// TwinCAT 3 PLC project RobustSolutionFramework
// Title: RobustSolution
// Company: BATW
// Author: BATW
// ProjectVersion: 1.0.0.1
// ProgramVersion: 3.1.4026.24
// libraries:
//   Tc2_MC2, * (Beckhoff Automation GmbH)
//   Tc2_Standard, * (Beckhoff Automation GmbH)
//   Tc2_System, * (Beckhoff Automation GmbH)
//   Tc2_Utilities, * (Beckhoff Automation GmbH)
//   Tc3_JsonXml, * (Beckhoff Automation GmbH)
// project tree:
//   Configuration/DUTs/ E_AlarmOperator.TcDUT, E_ConfigDataType.TcDUT (not stored), E_ConfigValueError.TcDUT, E_LinkPhase.TcDUT, E_ModuleType.TcDUT (not stored), T_ModuleTypeName.TcDUT, E_VariableAccess.TcDUT (not stored), ST_ConfigRawValue.TcDUT, ST_ReferenceBindingFileConfig.TcDUT (not stored), ST_ConfigAlarmInfo.TcDUT, ST_ConfigVariableInfo.TcDUT, ST_RuntimeAlarmBinding.TcDUT, ST_RuntimeVariableBinding.TcDUT, ST_LinkVariableNode.TcDUT (not stored), ST_MappingFileConfig.TcDUT (not stored), ST_ModuleFileConfig.TcDUT (not stored), ST_ModuleRuntimeConfig.TcDUT (not stored), ST_SystemFileConfig.TcDUT (not stored), ST_VariableLink.TcDUT
//   Configuration/POUs/ F_AlarmConditionMet.TcPOU (not stored), F_ConfigDataTypeSize.TcPOU (not stored), F_ConfigDataTypeToDescriptor.TcPOU, F_ConfigValueErrorMessage.TcPOU (not stored), FB_ConfigValueSnapshotReader.TcPOU, FB_ModuleTypeRegistry.TcPOU (not stored), FB_ReferenceManager.TcPOU (not stored), FB_ModuleReferenceBindingContext.TcPOU, FB_LinkVariableManager.TcPOU (not stored), FB_ModuleConfigurationManager.TcPOU (not stored), FB_ApplicationConfigRoot.TcPOU (not stored)
//   Configuration/Interfaces/ I_AdsSymbolProvider.TcIO (not stored), I_ModuleReferenceBindings.TcIO (not stored), I_ModuleConfigurationAdapter.TcIO (not stored), I_VariableNodeReader.TcIO (not stored)
//   DUTs/Contracts/Alarm/ E_Severity.TcDUT, ST_ExtAlarm.TcDUT
//   DUTs/Contracts/Descriptor/ E_DescriptorType.TcDUT, ST_ExtDescriptor.TcDUT (not stored)
//   DUTs/Contracts/System/ ST_SystemContext.TcDUT (not stored)
//   DUTs/Infrastructure/EL Modules/ ST_EL1889Ex.TcDUT (not stored), ST_EL2809Ex.TcDUT (not stored), ST_EL3602Ex.TcDUT (not stored)
//   DUTs/Infrastructure/ ST_ReserveForGetSymbolNameByAddrress.TcDUT
//   DUTs/Module/Alarm/ E_AlarmAckCommand.TcDUT (not stored), E_AlarmAckError.TcDUT (not stored), ST_AlarmAckRequest.TcDUT (not stored), ST_AlarmLifecycleState.TcDUT, ST_ModuleAlarmStatus.TcDUT (not stored)
//   DUTs/Module/Contract/ ST_ModuleCtrl.TcDUT, ST_ModuleDataStatus.TcDUT, ST_ModuleStatus.TcDUT, ST_ModuleVariableStatus.TcDUT (not stored), ST_Module_CtrlStatus_Base.TcDUT (not stored)
//   DUTs/Module/ServiceCoordination/ E_CompositeOwnershipState.TcDUT (not stored), E_ServiceCallSubmitResult.TcDUT (not stored), E_ServiceInternalCommandState.TcDUT, E_ServiceRegistrationError.TcDUT (not stored), ST_ServiceExecutionSnapshot.TcDUT (not stored), ST_ServiceRegistrationEntry.TcDUT (not stored)
//   DUTs/Service/Composite/ E_CompositeServiceErrorCode.TcDUT (not stored)
//   DUTs/Service/Contracts/ E_ServiceCompletionBehavior.TcDUT, ST_EmptyServiceParam.TcDUT, ST_ServiceContext.TcDUT, ST_ServiceCtrl.TcDUT (not stored), ST_ServiceDataStatus.TcDUT (not stored), ST_ServiceExecuteSubStateRecord.TcDUT, ST_ServiceExecuteSubStateStatus.TcDUT, ST_ServiceStatus.TcDUT
//   DUTs/Wafer Transfer/ E_MaterialOperateState.TcDUT, ST_MaterialContext.TcDUT, ST_WaferStatus.TcDUT
//   GVLs/ Param_Config.TcGVL
//   POUs/00_BaseUnit/Base/ FB_BaseUnit.TcPOU (not stored), T_ResourceOwnerId.TcDUT (not stored)
//   POUs/00_BaseUnit/ FB_Axis_BaseUnit.TcPOU (not stored)
//   POUs/00_BaseUnit/Interfaces/ I_Axis_BaseUnit.TcIO (not stored), I_BaseUnit.TcIO (not stored), I_ResourceLock.TcIO
//   POUs/10_Module/ FB_ModuleAlarmManager.TcPOU (not stored), FB_ModuleBase.TcPOU (not stored), FB_ServiceCoordinator.TcPOU, FB_ServiceCaller.TcPOU (not stored)
//   POUs/20_Service/ E_FrameworkServiceErrorCode.TcDUT, FB_CompositeServiceBase.TcPOU, FB_ServiceBase.TcPOU
//   POUs/20_Service/Material Service/ E_SetMaterialCmdType.TcDUT, FB_SetMaterialService.TcPOU, ST_MaterialParam.TcDUT
//   POUs/ FB_UtcClock.TcPOU
//   POUs/30_PackML_Base/DUTs/ E_PackMLCommand.TcDUT (not stored), E_PackMLErrorID.TcDUT (not stored), E_PackMLHookResult.TcDUT (not stored), E_PackMLMode.TcDUT (not stored), E_PackMLState.TcDUT, ST_PML_Base_In.TcDUT, ST_PML_Base_Out.TcDUT, T_PackMLMode.TcDUT (not stored)
//   POUs/30_PackML_Base/ FB_PackMLBase.TcPOU (not stored), FB_PackMLModeSet.TcPOU
//   POUs/30_PackML_Base/Utilities/ F_PackMLCommandToString.TcPOU (not stored), F_PackMLErrorIDToString.TcPOU (not stored), F_PackMLModeToString.TcPOU (not stored), F_PackMLStateToString.TcPOU (not stored)
// real-time tasks:
//   TASK UnitTest Task: cycle T#10ms, priority 21, ADS port 351
//   TASK DemoProject Task: cycle T#10ms, priority 22, ADS port 352
// motion (NC):
//   TASK NC-Task 1 SAF: cycle T#2ms, priority 4, ADS port 501
//   TASK NC-Task 1 SVB: cycle T#10ms, priority 8, ADS port 511
//   AXIS Axis 1 (id 1)
//     OtherSettings: AllowMotionCmdToSlave=true
//     encoder EncType=1
//     drive DrvType=5
//       Analog: TorqueSetpointScale=10, ScaleFactorActTorque=0.1
//       TimeComp: TaskDelayCycles=1
//     controller CtrType=1
//       CtrPara: PriorControlFactor=1
//         Observer: BandWidth=20
//   AXIS Axis 2 (id 2)
//     OtherSettings: AllowMotionCmdToSlave=true
//     encoder EncType=1
//     drive DrvType=5
//       Analog: TorqueSetpointScale=10, ScaleFactorActTorque=0.1
//       TimeComp: TaskDelayCycles=1
//     controller CtrType=1
//       CtrPara: PriorControlFactor=1
//         Observer: BandWidth=20
// variable links:
//   RobustSolutionDemoProject/RobustSolutionDemoProject Instance <-> NC-Task 1 SAF/Axes/Axis 1
//     PlcTask Inputs/GVL_IO.NC_Axis1._Axis.NcToPlc <-> Outputs/ToPlc
//     PlcTask Outputs/GVL_IO.NC_Axis1._Axis.PlcToNc <-> Inputs/FromPlc
//   RobustSolutionDemoProject/RobustSolutionDemoProject Instance <-> NC-Task 1 SAF/Axes/Axis 2
//     PlcTask Inputs/GVL_IO.NC_Axis2._Axis.NcToPlc <-> Outputs/ToPlc
//     PlcTask Outputs/GVL_IO.NC_Axis2._Axis.PlcToNc <-> Inputs/FromPlc

// ---- Configuration/DUTs/E_AlarmOperator.TcDUT
{attribute 'qualified_only'}
{attribute 'strict'}
{attribute 'to_string'}
TYPE E_AlarmOperator :
(
	Invalid := 0,
    GreaterThan,
    LessThan,
    Equal,
    GreaterOrEqual,
    LessOrEqual
);
END_TYPE

// ---- Configuration/DUTs/E_ConfigValueError.TcDUT
{attribute 'qualified_only'}
{attribute 'strict'}
{attribute 'to_string'}
TYPE E_ConfigValueError :
(
	None := 0,
	// FB_ConfigValueSnapshotReader cannot access the injected node reader.
	ReaderUnavailable := 16#7100,
	// The configured VariableList and AlarmList exceed the snapshot capacity.
	SourceCapacityExceeded := 16#7101,
	// FB_LinkVariableManager received an unknown or expired opaque handle.
	InvalidNodeHandle := 16#7201,
	// The registered node cannot be used as a configured value source.
	NodeReadNotAllowed := 16#7202,
	// The registered node no longer has a valid data address.
	InvalidNodeAddress := 16#7203,
	// Config metadata and registered node metadata do not describe the same type.
	NodeDataTypeMismatch := 16#7204,
	// The registered size is zero or exceeds ST_ConfigRawValue.Data.
	InvalidNodeSize := 16#7205
)UDINT;
END_TYPE

// ---- Configuration/DUTs/E_LinkPhase.TcDUT
{attribute 'qualified_only'}
{attribute 'strict'}
TYPE E_LinkPhase :
(
	InputToModule := 1,
	ModuleToOutput
);
END_TYPE

// ---- Configuration/DUTs/T_ModuleTypeName.TcDUT
TYPE T_ModuleTypeName : STRING(16);
END_TYPE

// ---- Configuration/DUTs/ST_ConfigRawValue.TcDUT
{attribute 'pack_mode' := '1'}
TYPE ST_ConfigRawValue :
STRUCT
	Data : ARRAY[0..Param_Config.MaxConfigValueSize - 1] OF BYTE;
END_STRUCT
END_TYPE

// ---- Configuration/DUTs/ST_ConfigAlarmInfo.TcDUT
TYPE ST_ConfigAlarmInfo :
STRUCT
	Source : STRING(255);
	DataType : E_ConfigDataType;
	Operator : E_AlarmOperator;
	Threshold : LREAL;
	Tolerance : LREAL;
	MainErrorId : UDINT;
	SourceErrorId : UDINT;
	Message : STRING(80);
	Severity : E_Severity;
END_STRUCT
END_TYPE

// ---- Configuration/DUTs/ST_ConfigVariableInfo.TcDUT
TYPE ST_ConfigVariableInfo :
STRUCT
	Source : STRING(255);
	Id : UDINT;
	Name : STRING(30);
	Unit : STRING(10);
	DataType : E_ConfigDataType;
END_STRUCT
END_TYPE

// ---- Configuration/DUTs/ST_RuntimeAlarmBinding.TcDUT
TYPE ST_RuntimeAlarmBinding :
STRUCT
	Definition : ST_ConfigAlarmInfo;
	NodeHandle : UINT;
END_STRUCT
END_TYPE

// ---- Configuration/DUTs/ST_RuntimeVariableBinding.TcDUT
TYPE ST_RuntimeVariableBinding :
STRUCT
	Definition : ST_ConfigVariableInfo;
	NodeHandle : UINT;
END_STRUCT
END_TYPE

// ---- Configuration/DUTs/ST_VariableLink.TcDUT
TYPE ST_VariableLink :
STRUCT
	SourceAddress : PVOID;
	TargetAddress : PVOID;
	SourceSize : UDINT;
	TargetSize : UDINT;
	SourceDataType : E_ConfigDataType;
	TargetDataType : E_ConfigDataType;
	Phase : E_LinkPhase;
	HasTransform : BOOL;
	Scale : LREAL;
	Offset : LREAL;
END_STRUCT
END_TYPE

// ---- DUTs/Contracts/Alarm/E_Severity.TcDUT
{attribute 'qualified_only'}
{attribute 'strict'}
{attribute 'to_string'}
TYPE E_Severity :
(
	Alarm := 1,
	Warning
);
END_TYPE

// ---- DUTs/Contracts/Alarm/ST_ExtAlarm.TcDUT
TYPE ST_ExtAlarm :
STRUCT
	ModuleId : UDINT;
	ServiceId : UDINT;
	MainErrorId : UDINT;
	SourceErrorId : UDINT;
	Message : STRING;
	Path : STRING(255);
	Severity : E_Severity;
	DateTime : STRING(20);	// First occurrence of the current alarm lifecycle. ex: YYYYMMDDHHMMSSUUU
	Active : BOOL;
	Acknowledged : BOOL;
	OccurrenceCount : UDINT;
END_STRUCT
END_TYPE

// ---- DUTs/Contracts/Descriptor/E_DescriptorType.TcDUT
{attribute 'qualified_only'}
{attribute 'strict'}
{attribute 'to_string'}
TYPE E_DescriptorType :
(
	Integer_32bit := 1,	// TwinCAT DINT, CSharp int
	Float_32bit,		// TwinCAT REAL, CSharp float
	String_80byte,
	DateTime,	// ex: YYYYMMDDHHMMSSUU
	Boolean,
	Unsigned_32bit,
	Float_64bit
);
END_TYPE

// ---- DUTs/Infrastructure/ST_ReserveForGetSymbolNameByAddrress.TcDUT
TYPE ST_ReserveForGetSymbolNameByAddrress :
STRUCT
	//If structures with a single variable are used, the data type cannot be read correctly using this method.
	//The size and address information cannot be used to distinguish between the structure itself and the individual variables.
	//https://infosys.beckhoff.com/content/1033/tcplclib_tc3_jsonxml/4220928907.html?id=4536537886268406375
	_Reserve : BOOL;
END_STRUCT
END_TYPE

// ---- DUTs/Module/Alarm/ST_AlarmLifecycleState.TcDUT
TYPE ST_AlarmLifecycleState :
STRUCT
	Latched : BOOL;
	PreviousActive : BOOL;
	SeenThisCycle : BOOL;
	Alarm : ST_ExtAlarm;
END_STRUCT
END_TYPE

// ---- DUTs/Module/Contract/ST_ModuleCtrl.TcDUT
TYPE ST_ModuleCtrl :
STRUCT
	RequestId : UDINT;
	PackMLIn : ST_PML_Base_In;
	
	AlarmAckRequest : ST_AlarmAckRequest;
END_STRUCT
END_TYPE

// ---- DUTs/Module/Contract/ST_ModuleDataStatus.TcDUT
TYPE ST_ModuleDataStatus :
STRUCT
	PublishedCount : UINT;
	Overflow : BOOL;
	DuplicateId : UDINT;
END_STRUCT
END_TYPE

// ---- DUTs/Module/Contract/ST_ModuleStatus.TcDUT
TYPE ST_ModuleStatus :
STRUCT
	ModuleId : UDINT;
	Enabled : BOOL;
	IsControlSourceAlive : BOOL;
	ModuleType : STRING(16);
	
	ResponseId : UDINT;
	PackMLOut : ST_PML_Base_Out;
	
	Alarm : ST_ModuleAlarmStatus;
	
	Data : ST_ModuleDataStatus;
	Variable : ST_ModuleVariableStatus;
	
	// Array index is storage only; EndpointId is the external identity.
	WaferStatusList : ARRAY [1..Param_Config.MaxTransferEndpoint] OF ST_WaferStatus;
END_STRUCT
END_TYPE

// ---- DUTs/Module/ServiceCoordination/E_ServiceInternalCommandState.TcDUT
{attribute 'qualified_only'}
{attribute 'strict'}
{attribute 'to_string'}
TYPE E_ServiceInternalCommandState :
(
	None := 0,
	Queued := 1,
	RequestHigh := 2,
	Accepted := 3,
	Rejected := 4,
	Cancelled := 5
) UDINT;
END_TYPE

// ---- DUTs/Service/Contracts/E_ServiceCompletionBehavior.TcDUT
{attribute 'qualified_only'}
{attribute 'strict'}
{attribute 'to_string'}
TYPE E_ServiceCompletionBehavior :
(
	Unknown := 0,
	NaturalCompletion := 1,
	ExecuteUntilExternalStop := 2
) UDINT;
END_TYPE

// ---- DUTs/Service/Contracts/ST_EmptyServiceParam.TcDUT
TYPE ST_EmptyServiceParam :
STRUCT
	bDummyValue : BOOL;	// To avoid 0 size check error during Service Coordinator Registration
END_STRUCT
END_TYPE

// ---- DUTs/Service/Contracts/ST_ServiceContext.TcDUT
TYPE ST_ServiceContext :
STRUCT
	ModuleId : UDINT;
	// UTC timestamp formatted as YYYYMMDDHHMMSSUUU.
	UtcDateTime : STRING(20);
END_STRUCT
END_TYPE

// ---- DUTs/Service/Contracts/ST_ServiceExecuteSubStateRecord.TcDUT
TYPE ST_ServiceExecuteSubStateRecord :
STRUCT
	Step : UDINT;
	Name : STRING(80);
	// UTC timestamp formatted as YYYYMMDDHHMMSSUUU.
	StartTimestamp : STRING(20);
	// Empty while this occurrence is still active.
	EndTimestamp : STRING(20);
END_STRUCT
END_TYPE

// ---- DUTs/Service/Contracts/ST_ServiceExecuteSubStateStatus.TcDUT
TYPE ST_ServiceExecuteSubStateStatus :
STRUCT
	// Zero whenever the Service is not executing or exposes no substate.
	CurrentStep : UDINT;
	RecordCount : UINT;
	// The first records are preserved when capacity is exhausted.
	Overflow : BOOL;
	Records : ARRAY[1..Param_Config.MaxExecuteSubStateRecords] OF ST_ServiceExecuteSubStateRecord;
END_STRUCT
END_TYPE

// ---- DUTs/Service/Contracts/ST_ServiceStatus.TcDUT
TYPE ST_ServiceStatus :
STRUCT
	ResponseId : UDINT;
	PackMLOut : ST_PML_Base_Out;
	ExecuteSubState : ST_ServiceExecuteSubStateStatus;
	CompletionBehavior : E_ServiceCompletionBehavior;
	ServiceId : UDINT;
	ErrorList : ARRAY[1..Param_Config.MaxServiceError] OF ST_ExtAlarm;
	Data : ST_ServiceDataStatus;
END_STRUCT
END_TYPE

// ---- DUTs/Wafer Transfer/E_MaterialOperateState.TcDUT
{attribute 'qualified_only'}
{attribute 'strict'}
{attribute 'to_string'}
TYPE E_MaterialOperateState :
(
	NotApplicable := 0,
	Pending,
	Processing,
	Completed,
	Failed
);
END_TYPE

// ---- DUTs/Wafer Transfer/ST_MaterialContext.TcDUT
TYPE ST_MaterialContext :
STRUCT
	Id : STRING(80);
	OperationState : E_MaterialOperateState;
	// Add other information of wafer...
END_STRUCT
END_TYPE

// ---- DUTs/Wafer Transfer/ST_WaferStatus.TcDUT
TYPE ST_WaferStatus :
STRUCT
	// Managed by module
	// Non-zero and unique within one Module; array index is storage only.
	EndpointId : UDINT;
	EndpointName : STRING(80);
	MaterialContext : ST_MaterialContext;
END_STRUCT
END_TYPE

// ---- POUs/20_Service/E_FrameworkServiceErrorCode.TcDUT
{attribute 'qualified_only'}
{attribute 'strict'}
{attribute 'to_string'}
TYPE E_FrameworkServiceErrorCode :
(
	// Set material service
	None := 0,
	SetMaterial_InvalidCmd := 900,
	SetMaterial_TaEpIdRequired := 901,
	SetMaterial_TaEpNotFound := 902,
	SetMaterial_DuplicateTaEpId := 903
) UDINT;
END_TYPE

// ---- POUs/20_Service/Material Service/E_SetMaterialCmdType.TcDUT
{attribute 'qualified_only'}
{attribute 'strict'}
{attribute 'to_string'}
TYPE E_SetMaterialCmdType :
(
	Modify:= 1,
	Clear,
	ClearAll
);
END_TYPE

// ---- POUs/20_Service/Material Service/ST_MaterialParam.TcDUT
TYPE ST_MaterialParam :
STRUCT
	CmdType : E_SetMaterialCmdType;
	TargetEndpointId : UDINT;
	
	// Material context
	MaterialId : STRING(80);
	MaterialOperateState : E_MaterialOperateState;
END_STRUCT
END_TYPE

// ---- POUs/30_PackML_Base/DUTs/E_PackMLState.TcDUT
{attribute 'qualified_only'}
TYPE E_PackMLState :
(
	Undefined		:= 0,
	Clearing		:= 1,
	Stopped			:= 2,
	Starting		:= 3,
	Idle			:= 4,
	Suspended		:= 5,
	Execute			:= 6,
	Stopping		:= 7,
	Aborting		:= 8,
	Aborted			:= 9,
	Holding			:= 10,
	Held			:= 11,
	Unholding		:= 12,
	Suspending		:= 13,
	Unsuspending	:= 14,
	Resetting		:= 15,
	Completing		:= 16,
	Complete		:= 17
);
END_TYPE

// ---- POUs/30_PackML_Base/DUTs/ST_PML_Base_In.TcDUT
TYPE ST_PML_Base_In :
STRUCT
	eCommand				: E_PackMLCommand := E_PackMLCommand.None;
	bCommandChangeRequest	: BOOL;
	eMode					: T_PackMLMode := E_PackMLMode.Unknown;
	bModeChangeRequest	: BOOL;
END_STRUCT
END_TYPE

// ---- POUs/30_PackML_Base/DUTs/ST_PML_Base_Out.TcDUT
TYPE ST_PML_Base_Out :
STRUCT
	eStateCurrent		: E_PackMLState := E_PackMLState.Undefined;
	eStatePrevious		: E_PackMLState := E_PackMLState.Undefined;
	eModeCurrent		: T_PackMLMode := E_PackMLMode.Unknown;
	eModePrevious		: T_PackMLMode := E_PackMLMode.Unknown;

	bCommandAccepted	: BOOL;
	bCommandRejected	: BOOL;
	eStateErrorID		: E_PackMLErrorID := E_PackMLErrorID.NoError;

	bModeChanged		: BOOL;
	bModeChangeRejected	: BOOL;
	eModeErrorID		: E_PackMLErrorID := E_PackMLErrorID.NoError;
END_STRUCT
END_TYPE

// ---- GVLs/Param_Config.TcGVL
{attribute 'qualified_only'}
VAR_GLOBAL CONSTANT
	MaxModuleVariable : UINT := 100;	// Num of SVID
	MaxConfiguredAlarmsPerModule : UINT := 30;	// Num of configured ALIDs.
	MaxHookAlarmsPerModule : UINT := 30;		// Reserved capacity for Module Hook alarms.
	MaxServiceAlarmsPerModule : UINT := 40;		// Reserved capacity for aggregated Service errors.
	MaxPublishedModuleAlarms : UINT := MaxConfiguredAlarmsPerModule + MaxHookAlarmsPerModule + MaxServiceAlarmsPerModule;
	MaxModuleAlarm : UINT := MaxPublishedModuleAlarms;	// Compatibility alias for existing consumers.
	MaxServiceError : UINT := 10;		// Num of Service Error per round
	MaxServiceData : UINT := 30;		// Num of persistent Data descriptors per Service
	MaxExecuteSubStateRecords : UINT := 30;	// Chronological Execute substate occurrences retained per Service run.
	MaxServicesPerModule : UINT := 100;	// Maximum number of Services registered by one Module.
	MaxCompositeDependencies : UINT := 10;	// Maximum number of child Services declared by one Composite Service.
	MaxModuleData : UINT := 50;			// Num of DVID
	MaxTransferEndpoint : UINT := 2;	// Num of wafer transfer port
	MaxProcessStation : UINT := 4;		// Num of wafer process station
	ModuleHeartbeat_Timeout : TIME := T#10S;

	// Runtime configuration limits. They also bound PLC memory and local snapshot work.
	MaxModuleTypes : UINT := 8;

	// Module type capacities bound type-specific runtime arrays.
	MaxModulePerType : UINT := 6;

	// Total config capacity is the compile-time sum of every supported Module type capacity.
	MaxTotalConfiguredModules : UINT := MaxModulePerType * MaxModuleTypes;

	// Variable mapping
	MaxModuleMappings : UINT := 256;
	MaxConfigVariableNodes : UINT := 512;

	// Reference binding
	MaxModuleReferences : UINT := 50;
	MaxConfigReferenceNodes : UINT := 100;

	// Registered-node snapshots used by configured VariableList and AlarmList.
	MaxConfiguredValueSources : UINT := MaxModuleVariable + MaxConfiguredAlarmsPerModule;
	MaxConfigValueSize : UINT := 81; // STRING(80), including the terminating zero.

	// System config
	ConfigSchemaVersion : UDINT := 4;
	ModuleConfigFilePath : STRING(255) := 'C:\ProgramData\RobustSolution\module-config.json';
END_VAR

// ---- POUs/00_BaseUnit/Interfaces/I_ResourceLock.TcIO
INTERFACE I_ResourceLock EXTENDS I_BaseUnit

METHOD M_AcquireResource : BOOL
VAR_INPUT
	OwnerId : T_ResourceOwnerId;
END_VAR
END_METHOD

METHOD M_IsResourceOwner : BOOL
VAR_INPUT
	OwnerId : T_ResourceOwnerId;
END_VAR
END_METHOD

METHOD M_ReleaseResource : BOOL
VAR_INPUT
	OwnerId : T_ResourceOwnerId;
END_VAR
END_METHOD

END_INTERFACE

// ---- Configuration/POUs/F_ConfigDataTypeToDescriptor.TcPOU
FUNCTION F_ConfigDataTypeToDescriptor : E_DescriptorType
VAR_INPUT
	DataType : E_ConfigDataType;
END_VAR

CASE DataType OF
	E_ConfigDataType.Boolean:
		F_ConfigDataTypeToDescriptor := E_DescriptorType.Boolean;
	E_ConfigDataType.Integer32:
		F_ConfigDataTypeToDescriptor := E_DescriptorType.Integer_32bit;
	E_ConfigDataType.UnsignedInteger32:
		F_ConfigDataTypeToDescriptor := E_DescriptorType.Unsigned_32bit;
	E_ConfigDataType.Float32:
		F_ConfigDataTypeToDescriptor := E_DescriptorType.Float_32bit;
	E_ConfigDataType.Float64:
		F_ConfigDataTypeToDescriptor := E_DescriptorType.Float_64bit;
	E_ConfigDataType.String80:
		F_ConfigDataTypeToDescriptor := E_DescriptorType.String_80byte;
ELSE
	F_ConfigDataTypeToDescriptor := E_DescriptorType.String_80byte;
END_CASE

END_FUNCTION

// ---- Configuration/POUs/FB_ConfigValueSnapshotReader.TcPOU
FUNCTION_BLOCK FB_ConfigValueSnapshotReader
VAR_INPUT
	RuntimeConfig : REFERENCE TO ST_ModuleRuntimeConfig;
	VariableNodeReader : I_VariableNodeReader;
END_VAR
VAR_OUTPUT
	Ready : BOOL;
	Error : BOOL;
	ErrorCode : E_ConfigValueError;
	ErrorMessage : STRING(255);
	ErrorSource : STRING(255);
END_VAR
VAR
	_SourceCount : UINT;
	_SourceTypes : ARRAY[1..Param_Config.MaxConfiguredValueSources] OF E_ConfigDataType;
	_Values : ARRAY[1..Param_Config.MaxConfiguredValueSources] OF ST_ConfigRawValue;
	_ValueValid : ARRAY[1..Param_Config.MaxConfiguredValueSources] OF BOOL;

END_VAR
VAR_TEMP
	_nIndex : UINT;
	_nSource : UINT;
	_eReadError : E_ConfigValueError;
END_VAR

Ready := FALSE;
Error := FALSE;
ErrorCode := E_ConfigValueError.None;
ErrorMessage := '';
ErrorSource := '';
_SourceCount := 0;

IF NOT __ISVALIDREF(RuntimeConfig) THEN
	RETURN;
END_IF
IF NOT RuntimeConfig.Enabled OR NOT RuntimeConfig.Valid THEN
	RETURN;
END_IF
IF VariableNodeReader = 0 THEN
	M_SetFirstError(
		ErrorCodeValue := E_ConfigValueError.ReaderUnavailable,
		SourceName := '');
	RETURN;
END_IF

_SourceCount := RuntimeConfig.VariableCount + RuntimeConfig.AlarmCount;
IF _SourceCount > Param_Config.MaxConfiguredValueSources THEN
	M_SetFirstError(
		ErrorCodeValue := E_ConfigValueError.SourceCapacityExceeded,
		SourceName := '');
	RETURN;
END_IF

MEMSET(ADR(_SourceTypes), 0, SIZEOF(_SourceTypes));
MEMSET(ADR(_ValueValid), 0, SIZEOF(_ValueValid));

FOR _nIndex := 1 TO RuntimeConfig.VariableCount DO
	_nSource := _nIndex;
	_SourceTypes[_nSource] := RuntimeConfig.VariableBindings[_nIndex].Definition.DataType;
	_ValueValid[_nSource] := VariableNodeReader.M_ReadNode(
		NodeHandle := RuntimeConfig.VariableBindings[_nIndex].NodeHandle,
		ExpectedDataType := _SourceTypes[_nSource],
		Value := _Values[_nSource],
		ErrorCode => _eReadError);
	IF NOT _ValueValid[_nSource] AND NOT Error THEN
		M_SetFirstError(
			ErrorCodeValue := _eReadError,
			SourceName := RuntimeConfig.VariableBindings[_nIndex].Definition.Source);
	END_IF
END_FOR

FOR _nIndex := 1 TO RuntimeConfig.AlarmCount DO
	_nSource := RuntimeConfig.VariableCount + _nIndex;
	_SourceTypes[_nSource] := RuntimeConfig.AlarmBindings[_nIndex].Definition.DataType;
	_ValueValid[_nSource] := VariableNodeReader.M_ReadNode(
		NodeHandle := RuntimeConfig.AlarmBindings[_nIndex].NodeHandle,
		ExpectedDataType := _SourceTypes[_nSource],
		Value := _Values[_nSource],
		ErrorCode => _eReadError);
	IF NOT _ValueValid[_nSource] AND NOT Error THEN
		M_SetFirstError(
			ErrorCodeValue := _eReadError,
			SourceName := RuntimeConfig.AlarmBindings[_nIndex].Definition.Source);
	END_IF
END_FOR

Ready := NOT Error;

METHOD PUBLIC M_GetLReal : LREAL
VAR_INPUT
	SourceIndex : UINT;
END_VAR
VAR_OUTPUT
	Valid : BOOL;
END_VAR
VAR
	pBool : POINTER TO BOOL;
	pDInt : POINTER TO DINT;
	pUDInt : POINTER TO UDINT;
	pReal : POINTER TO REAL;
	pLReal : POINTER TO LREAL;
END_VAR
Valid := FALSE;
M_GetLReal := 0.0;
IF NOT Ready OR (SourceIndex < 1) OR (SourceIndex > _SourceCount)
	OR NOT _ValueValid[SourceIndex] THEN
	RETURN;
END_IF

CASE _SourceTypes[SourceIndex] OF
	E_ConfigDataType.Boolean:
		pBool := ADR(_Values[SourceIndex].Data);
		IF pBool^ THEN M_GetLReal := 1.0; END_IF
	E_ConfigDataType.Integer32:
		pDInt := ADR(_Values[SourceIndex].Data);
		M_GetLReal := DINT_TO_LREAL(pDInt^);
	E_ConfigDataType.UnsignedInteger32:
		pUDInt := ADR(_Values[SourceIndex].Data);
		M_GetLReal := UDINT_TO_LREAL(pUDInt^);
	E_ConfigDataType.Float32:
		pReal := ADR(_Values[SourceIndex].Data);
		M_GetLReal := REAL_TO_LREAL(pReal^);
	E_ConfigDataType.Float64:
		pLReal := ADR(_Values[SourceIndex].Data);
		M_GetLReal := pLReal^;
ELSE
	RETURN;
END_CASE
Valid := TRUE;
END_METHOD

METHOD PUBLIC M_GetValueString : STRING(80)
VAR_INPUT
	SourceIndex : UINT;
END_VAR
VAR_OUTPUT
	Valid : BOOL;
END_VAR
VAR
	pBool : POINTER TO BOOL;
	pDInt : POINTER TO DINT;
	pUDInt : POINTER TO UDINT;
	pReal : POINTER TO REAL;
	pLReal : POINTER TO LREAL;
	sValue : STRING(80);
END_VAR
Valid := FALSE;
M_GetValueString := '';
IF NOT Ready OR (SourceIndex < 1) OR (SourceIndex > _SourceCount) THEN
	RETURN;
END_IF

// TwinCAT 的普通 OR 不保證短路求值
IF NOT _ValueValid[SourceIndex] THEN
	RETURN;
END_IF

CASE _SourceTypes[SourceIndex] OF
	E_ConfigDataType.Boolean:
		pBool := ADR(_Values[SourceIndex].Data);
		sValue := BOOL_TO_STRING(pBool^);
	E_ConfigDataType.Integer32:
		pDInt := ADR(_Values[SourceIndex].Data);
		sValue := DINT_TO_STRING(pDInt^);
	E_ConfigDataType.UnsignedInteger32:
		pUDInt := ADR(_Values[SourceIndex].Data);
		sValue := UDINT_TO_STRING(pUDInt^);
	E_ConfigDataType.Float32:
		pReal := ADR(_Values[SourceIndex].Data);
		sValue := REAL_TO_STRING(pReal^);
	E_ConfigDataType.Float64:
		pLReal := ADR(_Values[SourceIndex].Data);
		sValue := LREAL_TO_STRING(pLReal^);
	E_ConfigDataType.String80:
		MEMCPY(ADR(sValue), ADR(_Values[SourceIndex].Data), SIZEOF(sValue));
ELSE
	RETURN;
END_CASE
M_GetValueString := sValue;
Valid := TRUE;
END_METHOD

METHOD PRIVATE M_SetFirstError
VAR_INPUT
	ErrorCodeValue : E_ConfigValueError;
	SourceName : STRING(255);
END_VAR
IF Error THEN
	RETURN;
END_IF

Error := TRUE;
ErrorCode := ErrorCodeValue;
ErrorMessage := F_ConfigValueErrorMessage(ErrorCode := ErrorCodeValue);
ErrorSource := SourceName;
END_METHOD

END_FUNCTION_BLOCK

// ---- Configuration/POUs/FB_ModuleReferenceBindingContext.TcPOU
FUNCTION_BLOCK FB_ModuleReferenceBindingContext IMPLEMENTS I_ModuleReferenceBindings
VAR_OUTPUT
	Error : BOOL;
	ErrorMessage : STRING(255);
END_VAR
VAR
	_Names : ARRAY[1..Param_Config.MaxModuleReferences] OF STRING(80);
	_SourceNames : ARRAY[1..Param_Config.MaxModuleReferences] OF STRING(255);
	_Consumed : ARRAY[1..Param_Config.MaxModuleReferences] OF BOOL;
	_ReferenceManager : REFERENCE TO FB_ReferenceManager;
	_Count : UINT;
	_Active : BOOL;
	_ModuleSymbol : STRING(255);
	_JsonDataType : FB_JsonReadWriteDataType;
END_VAR

METHOD PUBLIC M_Begin : BOOL
VAR_IN_OUT CONSTANT
	ModuleConfig : ST_ModuleFileConfig;
END_VAR
VAR_IN_OUT
	ReferenceManager : FB_ReferenceManager;
END_VAR
VAR
	nItem : UINT;
	nOther : UINT;
END_VAR
M_Begin := FALSE;
M_Clear();

IF ModuleConfig.ReferenceCount > Param_Config.MaxModuleReferences THEN
	Error := TRUE;
	ErrorMessage := 'Module reference capacity was exceeded.';
	RETURN;
END_IF

FOR nItem := 1 TO ModuleConfig.ReferenceCount DO
	IF (ModuleConfig.References[nItem].Name = '') OR (ModuleConfig.References[nItem].Source = '') THEN
		Error := TRUE;
		ErrorMessage := 'Every Module reference requires a name and source.';
		RETURN;
	END_IF

	IF nItem > 1 THEN
		FOR nOther := 1 TO nItem - 1 DO
			IF ModuleConfig.References[nOther].Name = ModuleConfig.References[nItem].Name THEN
				Error := TRUE;
				ErrorMessage := CONCAT('Duplicate Module reference name: ', ModuleConfig.References[nItem].Name);
				RETURN;
			END_IF
		END_FOR
	END_IF

	_Names[nItem] := ModuleConfig.References[nItem].Name;
	_SourceNames[nItem] := ModuleConfig.References[nItem].Source;
END_FOR

_Count := ModuleConfig.ReferenceCount;
_ReferenceManager REF= ReferenceManager;
_Active := TRUE;
M_Begin := TRUE;
END_METHOD

METHOD PUBLIC M_Clear
VAR
	nItem : UINT;
END_VAR
FOR nItem := 1 TO Param_Config.MaxModuleReferences DO
	_Names[nItem] := '';
	_SourceNames[nItem] := '';
	_Consumed[nItem] := FALSE;
END_FOR
_Count := 0;
_Active := FALSE;
_ModuleSymbol := '';
Error := FALSE;
ErrorMessage := '';
END_METHOD

METHOD PUBLIC M_End : BOOL
VAR
	nItem : UINT;
END_VAR
M_End := FALSE;
IF Error THEN
	RETURN;
END_IF
IF NOT _Active THEN
	Error := TRUE;
	ErrorMessage := 'No Module reference binding context is active.';
	RETURN;
END_IF

FOR nItem := 1 TO _Count DO
	IF NOT _Consumed[nItem] THEN
		Error := TRUE;
		ErrorMessage := CONCAT('Unknown Module reference name: ', _Names[nItem]);
		RETURN;
	END_IF
END_FOR

_Active := FALSE;
M_End := TRUE;
END_METHOD

METHOD PRIVATE M_Take : I_BaseUnit
VAR_INPUT
	Name : STRING(80);
	Required : BOOL;
END_VAR
VAR_OUTPUT
	Present : BOOL;
	TakeErrorMessage : STRING(255);
END_VAR
VAR
	nItem : UINT;
	BaseUnit : I_BaseUnit;
END_VAR
M_Take := 0;
Present := FALSE;
TakeErrorMessage := '';
IF Error THEN
	TakeErrorMessage := ErrorMessage;
	RETURN;
END_IF
IF NOT _Active THEN
	Error := TRUE;
	ErrorMessage := 'No Module reference binding context is active.';
	TakeErrorMessage := ErrorMessage;
	RETURN;
END_IF
IF Name = '' THEN
	Error := TRUE;
	ErrorMessage := 'A Module reference name is required.';
	TakeErrorMessage := ErrorMessage;
	RETURN;
END_IF

FOR nItem := 1 TO _Count DO
	IF _Names[nItem] = Name THEN
		IF _Consumed[nItem] THEN
			Error := TRUE;
			ErrorMessage := CONCAT('Module reference was taken more than once: ', Name);
			TakeErrorMessage := ErrorMessage;
			RETURN;
		END_IF
		IF NOT __ISVALIDREF(_ReferenceManager) THEN
			Error := TRUE;
			ErrorMessage := 'The Module reference source registry is unavailable.';
			TakeErrorMessage := ErrorMessage;
			RETURN;
		END_IF
		BaseUnit := _ReferenceManager.M_Resolve(Name := _SourceNames[nItem]);
		IF BaseUnit = 0 THEN
			Error := TRUE;
			ErrorMessage := CONCAT('Module reference source was not registered: ', _SourceNames[nItem]);
			TakeErrorMessage := ErrorMessage;
			RETURN;
		END_IF
		_Consumed[nItem] := TRUE;
		Present := TRUE;
		M_Take := BaseUnit;
		RETURN;
	END_IF
END_FOR

IF Required THEN
	Error := TRUE;
	ErrorMessage := CONCAT('Missing required Module reference: ', Name);
	TakeErrorMessage := ErrorMessage;
END_IF
END_METHOD

METHOD PUBLIC M_TakeOptional : I_BaseUnit
VAR_INPUT
	Port : ANY;
END_VAR
VAR_OUTPUT
	PortName : STRING(80);
	Present : BOOL;
	ErrorMessage : STRING(255);
END_VAR
M_TakeOptional := 0;
Present := FALSE;
IF NOT M_ResolvePortName(
	Port := Port,
	PortName => PortName,
	ResolveErrorMessage => ErrorMessage) THEN
	RETURN;
END_IF
M_TakeOptional := M_Take(
	Name := PortName,
	Required := FALSE,
	Present => Present,
	TakeErrorMessage => ErrorMessage);
END_METHOD

METHOD PUBLIC M_TakeRequired : I_BaseUnit
VAR_INPUT
	Port : ANY;
END_VAR
VAR_OUTPUT
	PortName : STRING(80);
	ErrorMessage : STRING(255);
END_VAR
VAR
	bPresent : BOOL;
END_VAR
M_TakeRequired := 0;
IF NOT M_ResolvePortName(
	Port := Port,
	PortName => PortName,
	ResolveErrorMessage => ErrorMessage) THEN
	RETURN;
END_IF
M_TakeRequired := M_Take(
	Name := PortName,
	Required := TRUE,
	Present => bPresent,
	TakeErrorMessage => ErrorMessage);
END_METHOD

METHOD PUBLIC M_SetModuleScope : BOOL
VAR_INPUT
	ModuleSymbol : STRING(255);
END_VAR
VAR_OUTPUT
	ErrorMessage : STRING(255);
END_VAR
M_SetModuleScope := FALSE;
ErrorMessage := '';
IF Error THEN
	ErrorMessage := THIS^.ErrorMessage;
	RETURN;
END_IF
IF NOT _Active THEN
	M_SetError(Message := 'No Module reference binding context is active.');
ELSIF _ModuleSymbol <> '' THEN
	M_SetError(Message := 'The Module reference scope was already set.');
ELSIF ModuleSymbol = '' THEN
	M_SetError(Message := 'A Module ADS symbol name is required for reference binding.');
ELSE
	_ModuleSymbol := ModuleSymbol;
	M_SetModuleScope := TRUE;
END_IF
IF Error THEN
	ErrorMessage := THIS^.ErrorMessage;
END_IF
END_METHOD

METHOD PRIVATE M_SetError
VAR_INPUT
	Message : STRING(255);
END_VAR
IF NOT Error THEN
	Error := TRUE;
	ErrorMessage := Message;
END_IF
END_METHOD

METHOD PRIVATE M_ResolvePortName : BOOL
VAR_INPUT
	Port : ANY;
END_VAR
VAR_OUTPUT
	PortName : STRING(80);
	ResolveErrorMessage : STRING(255);
END_VAR
VAR
	sSymbol : STRING(255);
	nPrefixLength : INT;
	nNameLength : INT;
	hrErrorCode : HRESULT;
END_VAR
M_ResolvePortName := FALSE;
PortName := '';
ResolveErrorMessage := '';
IF Error THEN
	ResolveErrorMessage := ErrorMessage;
	RETURN;
END_IF
IF NOT _Active THEN
	M_SetError(Message := 'No Module reference binding context is active.');
ELSIF _ModuleSymbol = '' THEN
	M_SetError(Message := 'Set the Module reference scope before taking a port.');
ELSIF (Port.pValue = 0) OR (Port.diSize <= 0) THEN
	M_SetError(Message := 'A reference port requires a valid variable address and positive size.');
END_IF
IF Error THEN
	ResolveErrorMessage := ErrorMessage;
	RETURN;
END_IF

// Inspect the caller's interface storage, even when its current value is zero.
// Never dereference Port.pValue or retain it after this initialization call.
sSymbol := _JsonDataType.GetSymbolNameByAddress(
	nData := DINT_TO_UDINT(Port.diSize),
	pData := Port.pValue,
	hrErrorCode => hrErrorCode);
IF (hrErrorCode <> 0) OR (sSymbol = '') THEN
	M_SetError(Message := 'Cannot resolve the reference port ADS symbol name.');
ELSE
	nPrefixLength := LEN(_ModuleSymbol) + 1;
	IF LEN(sSymbol) <= nPrefixLength THEN
		M_SetError(Message := 'The reference port must be a member of the active Module instance.');
	ELSIF (LEFT(sSymbol, LEN(_ModuleSymbol)) <> _ModuleSymbol)
		OR (MID(sSymbol, 1, nPrefixLength) <> '.') THEN
		M_SetError(Message := CONCAT('Reference port belongs to a different Module scope: ', sSymbol));
	ELSE
		nNameLength := LEN(sSymbol) - nPrefixLength;
		IF nNameLength > 80 THEN
			M_SetError(Message := 'The relative reference port name exceeds 80 characters.');
		ELSE
			// Preserve the full relative path, including nested members and array indices.
			PortName := RIGHT(sSymbol, nNameLength);
			M_ResolvePortName := TRUE;
		END_IF
	END_IF
END_IF
IF Error THEN
	ResolveErrorMessage := ErrorMessage;
END_IF
END_METHOD

END_FUNCTION_BLOCK

// ---- POUs/10_Module/FB_ServiceCoordinator.TcPOU
FUNCTION_BLOCK FB_ServiceCoordinator
VAR
	_Entries : ARRAY[1..Param_Config.MaxServicesPerModule] OF ST_ServiceRegistrationEntry;
	_RegisteredCount : UINT;
	_RegistrationStarted : BOOL;
	_Sealed : BOOL;
	_RegistrationError : E_ServiceRegistrationError;
	_FailedServiceId : UDINT;
	_AllIdle : BOOL;
	_AllStopped : BOOL;
	_AllAborted : BOOL;
	_JsonDataType : FB_JsonReadWriteDataType;
END_VAR

PROPERTY PUBLIC FINAL AllAborted : BOOL
GET
AllAborted := _AllAborted;
END_GET
END_PROPERTY

PROPERTY PUBLIC FINAL AllIdle : BOOL
GET
AllIdle := _AllIdle;
END_GET
END_PROPERTY

PROPERTY PUBLIC FINAL AllStopped : BOOL
GET
AllStopped := _AllStopped;
END_GET
END_PROPERTY

PROPERTY PUBLIC FINAL FailedServiceId : UDINT
GET
FailedServiceId := _FailedServiceId;
END_GET
END_PROPERTY

METHOD PUBLIC FINAL M_BeginRegistration : BOOL
// 開啟一次性的 Service 註冊階段；必須先於 M_Register 與 M_Seal 呼叫。
// 成功時會清除舊登錄資料與彙總狀態；重複呼叫則留下 RegistrationAlreadyStarted 錯誤。
M_BeginRegistration := FALSE;
IF _RegistrationStarted THEN
	M_SetRegistrationError(Error := E_ServiceRegistrationError.RegistrationAlreadyStarted, ServiceId := 0);
	RETURN;
END_IF

// 重設 Coordinator 的註冊內容，但不允許用此方法重新開啟已經開始過的註冊流程。
MEMSET(ADR(_Entries), 0, SIZEOF(_Entries));
_RegisteredCount := 0;
_Sealed := FALSE;
_RegistrationError := E_ServiceRegistrationError.None;
_FailedServiceId := 0;
_AllIdle := FALSE;
_AllStopped := FALSE;
_AllAborted := FALSE;
_RegistrationStarted := TRUE;
M_BeginRegistration := TRUE;
END_METHOD

METHOD PRIVATE M_FindIndexByServiceId : UINT
VAR_INPUT
	ServiceId : UDINT;
END_VAR
VAR
	nIndex : UINT;
END_VAR
M_FindIndexByServiceId := 0;
IF ServiceId = 0 THEN RETURN; END_IF
FOR nIndex := 1 TO _RegisteredCount DO
	IF _Entries[nIndex].InUse AND (_Entries[nIndex].ServiceId = ServiceId) THEN
		M_FindIndexByServiceId := nIndex;
		RETURN;
	END_IF
END_FOR
END_METHOD

METHOD PUBLIC FINAL M_GetCompositeOwnershipState : E_CompositeOwnershipState
VAR_INPUT
	CompositeServiceId : UDINT;
END_VAR
VAR
	nIndex : UINT;
END_VAR
// 查詢 Composite Service 的 ownership 流程狀態。
// 找不到 Service 或目標不是 Composite 時回傳 None，呼叫端可將其視為無有效 ownership。
M_GetCompositeOwnershipState := E_CompositeOwnershipState.None;
nIndex := M_FindIndexByServiceId(ServiceId := CompositeServiceId);
IF (nIndex = 0) OR NOT _Entries[nIndex].IsComposite THEN RETURN; END_IF

// Pending 會在 M_PrepareCycle 中解析為 Owned、Rejected 或 Cancelled。
M_GetCompositeOwnershipState := _Entries[nIndex].OwnershipState;
END_METHOD

METHOD PUBLIC FINAL M_GetInternalCommandState : E_ServiceInternalCommandState
VAR_INPUT
	CallerServiceId : UDINT;
	TargetServiceId : UDINT;
END_VAR
VAR
	nCallerIndex : UINT;
	nTargetIndex : UINT;
END_VAR
// 查詢 Composite 對指定 dependency 所送內部命令的握手狀態。
// Caller、Target 或 dependency 關係無效時回傳 None，避免讀到其他 Service 的內部狀態。
M_GetInternalCommandState := E_ServiceInternalCommandState.None;
nCallerIndex := M_FindIndexByServiceId(ServiceId := CallerServiceId);
nTargetIndex := M_FindIndexByServiceId(ServiceId := TargetServiceId);
IF (nCallerIndex = 0) OR (nTargetIndex = 0) THEN RETURN; END_IF
IF NOT M_IsDeclaredDependency(CompositeIndex := nCallerIndex, TargetServiceId := TargetServiceId) THEN RETURN; END_IF

// ownership 已移轉時不公開舊狀態；Cancelled 例外保留，讓原 Caller 得知請求被取消。
IF (_Entries[nTargetIndex].CompositeOwnerServiceId <> CallerServiceId)
	AND (_Entries[nTargetIndex].InternalCommandState <> E_ServiceInternalCommandState.Cancelled) THEN RETURN; END_IF
M_GetInternalCommandState := _Entries[nTargetIndex].InternalCommandState;
END_METHOD

METHOD PUBLIC FINAL M_GetServiceSnapshotById : BOOL
VAR_INPUT
	ServiceId : UDINT;
END_VAR
VAR_OUTPUT
	Snapshot : ST_ServiceExecutionSnapshot;
END_VAR
VAR
	nIndex : UINT;
END_VAR
// 依 ServiceId 取得最近一次 M_ObserveCycle 保存的執行快照，而非即時讀取 Service 狀態。
// 查詢失敗或快照尚未建立時回傳 FALSE，並確保輸出 Snapshot 為零值。
M_GetServiceSnapshotById := FALSE;
MEMSET(ADR(Snapshot), 0, SIZEOF(Snapshot));
nIndex := M_FindIndexByServiceId(ServiceId := ServiceId);
IF nIndex = 0 THEN RETURN; END_IF

// Valid 只有在 M_ObserveCycle 至少觀察過該 Service 一次後才會成立。
Snapshot := _Entries[nIndex].ObservedSnapshot;
M_GetServiceSnapshotById := Snapshot.Valid;
END_METHOD

METHOD PUBLIC FINAL M_GetServiceStatusByIndex : BOOL
VAR_INPUT
	Index : UINT;
END_VAR
VAR_OUTPUT
	Status : ST_ServiceStatus;
END_VAR
VAR
	pStatus : POINTER TO ST_ServiceStatus;
END_VAR
// 以 1-based 註冊索引複製 Service 的即時 Status，供 Module 層彙整 alarm、data 與狀態。
// 索引或登錄儲存位置無效時回傳 FALSE，並將輸出 Status 清為零值。
M_GetServiceStatusByIndex := FALSE;
MEMSET(ADR(Status), 0, SIZEOF(Status));
IF (Index = 0) OR (Index > _RegisteredCount) THEN RETURN; END_IF
IF NOT _Entries[Index].InUse OR (_Entries[Index].StatusAddress = 0) THEN RETURN; END_IF

// StatusAddress 指向 M_Register 時提供的長期存在變數；此處只複製內容，不保留新指標。
pStatus := _Entries[Index].StatusAddress;
Status := pStatus^;
M_GetServiceStatusByIndex := TRUE;
END_METHOD

METHOD PRIVATE M_IsDeclaredDependency : BOOL
VAR_INPUT
	CompositeIndex : UINT;
	TargetServiceId : UDINT;
END_VAR
VAR
	nDependency : UINT;
	pDependencies : POINTER TO UDINT;
END_VAR
M_IsDeclaredDependency := FALSE;
IF (CompositeIndex = 0) OR (CompositeIndex > _RegisteredCount)
	OR NOT _Entries[CompositeIndex].IsComposite
	OR (_Entries[CompositeIndex].CompositeDependenciesAddress = 0) THEN RETURN; END_IF

pDependencies := _Entries[CompositeIndex].CompositeDependenciesAddress;
FOR nDependency := 1 TO _Entries[CompositeIndex].CompositeDependencyCount DO
	IF pDependencies[nDependency - 1] = TargetServiceId THEN
		M_IsDeclaredDependency := TRUE;
		RETURN;
	END_IF
END_FOR
END_METHOD

METHOD PUBLIC FINAL M_ObserveCycle
VAR
	nIndex : UINT;
	pStatus : POINTER TO ST_ServiceStatus;
END_VAR
// 每個 PLC scan 在所有 Service 執行完成後呼叫，用來保存本週期結果。
// Coordinator 未 Ready 或沒有已註冊 Service 時，所有彙總狀態維持 FALSE。
_AllIdle := FALSE;
_AllStopped := FALSE;
_AllAborted := FALSE;
IF NOT Ready OR (_RegisteredCount = 0) THEN RETURN; END_IF

// 先假設所有 Service 位於同一目標狀態，再逐筆以 AND 收斂彙總結果。
_AllIdle := TRUE;
_AllStopped := TRUE;
_AllAborted := TRUE;
FOR nIndex := 1 TO _RegisteredCount DO
	pStatus := _Entries[nIndex].StatusAddress;

	// 保存穩定快照，讓 Composite 在下一個控制週期查詢 ResponseId、PackML 與執行步驟。
	_Entries[nIndex].ObservedSnapshot.Valid := TRUE;
	_Entries[nIndex].ObservedSnapshot.ServiceId := _Entries[nIndex].ServiceId;
	_Entries[nIndex].ObservedSnapshot.ResponseId := pStatus^.ResponseId;
	_Entries[nIndex].ObservedSnapshot.PackMLOut := pStatus^.PackMLOut;
	_Entries[nIndex].ObservedSnapshot.ExecuteSubState := pStatus^.ExecuteSubState.CurrentStep;
	_Entries[nIndex].ObservedSnapshot.CompletionBehavior := pStatus^.CompletionBehavior;

	// 只有相同 RequestId 的回覆可完成內部命令；完成後要求 M_PrepareCycle 輸出一個低電位週期。
	IF (_Entries[nIndex].InternalCommandState = E_ServiceInternalCommandState.RequestHigh)
		AND (pStatus^.ResponseId = _Entries[nIndex].InternalRequestId) THEN
		IF pStatus^.PackMLOut.bCommandAccepted THEN
			_Entries[nIndex].InternalCommandState := E_ServiceInternalCommandState.Accepted;
			_Entries[nIndex].InternalRequestMustGoLow := TRUE;
		ELSIF pStatus^.PackMLOut.bCommandRejected THEN
			_Entries[nIndex].InternalCommandState := E_ServiceInternalCommandState.Rejected;
			_Entries[nIndex].InternalRequestMustGoLow := TRUE;
		END_IF
	END_IF
	// 同步更新 Module lifecycle 使用的 AllIdle、AllStopped 與 AllAborted。
	_AllIdle := _AllIdle AND (pStatus^.PackMLOut.eStateCurrent = E_PackMLState.Idle);
	_AllStopped := _AllStopped AND (pStatus^.PackMLOut.eStateCurrent = E_PackMLState.Stopped);
	_AllAborted := _AllAborted AND (pStatus^.PackMLOut.eStateCurrent = E_PackMLState.Aborted);
END_FOR
END_METHOD

METHOD PUBLIC FINAL M_PrepareCycle
VAR_INPUT
	ModuleInExecute : BOOL;
	ModuleCtrl : REFERENCE TO ST_ModuleCtrl;
END_VAR
VAR
	nIndex : UINT;
	pUpperCtrl : POINTER TO ST_ServiceCtrl;
	pEffectiveCtrl : POINTER TO ST_ServiceCtrl;
	bUpperCommandHigh : BOOL;
	bUpperModeHigh : BOOL;
	bNewStartRequest : BOOL;
END_VAR
// Resolve Composite ownership only while the Module can execute Services.
// Pending requests are cancelled outside Execute so they cannot leak into a later cycle.
IF Ready AND ModuleInExecute THEN
	M_ProcessOwnershipRequests();
ELSIF Ready THEN
	FOR nIndex := 1 TO _RegisteredCount DO
		IF _Entries[nIndex].OwnershipState = E_CompositeOwnershipState.Pending THEN
			_Entries[nIndex].OwnershipState := E_CompositeOwnershipState.Cancelled;
		END_IF
	END_FOR
END_IF

// Build the effective control input consumed by each registered Service.
FOR nIndex := 1 TO _RegisteredCount DO
	pUpperCtrl := _Entries[nIndex].UpperCtrlAddress;
	pEffectiveCtrl := _Entries[nIndex].EffectiveCtrlAddress;
	
	// A registration error makes all Service request signals inactive.
	IF NOT Ready THEN
		pEffectiveCtrl^.PackMLIn.bCommandChangeRequest := FALSE;
		pEffectiveCtrl^.PackMLIn.bModeChangeRequest := FALSE;
		CONTINUE;
	END_IF
	
	bUpperCommandHigh := pUpperCtrl^.PackMLIn.bCommandChangeRequest;
	bUpperModeHigh := pUpperCtrl^.PackMLIn.bModeChangeRequest;
	
	// Outside Module Execute, cancel Composite-issued requests and propagate only the
	// Module lifecycle commands that are valid for bringing every Service to a safe state.
	IF NOT ModuleInExecute THEN
		IF (_Entries[nIndex].InternalCommandState = E_ServiceInternalCommandState.Queued)
			OR (_Entries[nIndex].InternalCommandState = E_ServiceInternalCommandState.RequestHigh)
			OR _Entries[nIndex].InternalRequestMustGoLow THEN
			_Entries[nIndex].InternalCommandState := E_ServiceInternalCommandState.Cancelled;
			_Entries[nIndex].InternalRequestMustGoLow := FALSE;
		END_IF
		pEffectiveCtrl^.RequestId := ModuleCtrl.RequestId;
		pEffectiveCtrl^.PackMLIn := ModuleCtrl.PackMLIn;
		
		// Only Module lifecycle commands may control the registered Services.
		// Module Start and other commands must not become Service requests.
		IF (NOT pEffectiveCtrl^.PackMLIn.bCommandChangeRequest)
			OR ((pEffectiveCtrl^.PackMLIn.eCommand <> E_PackMLCommand.Stop)
				AND (pEffectiveCtrl^.PackMLIn.eCommand <> E_PackMLCommand.Abort)
				AND (pEffectiveCtrl^.PackMLIn.eCommand <> E_PackMLCommand.Clear)
				AND (pEffectiveCtrl^.PackMLIn.eCommand <> E_PackMLCommand.Reset)) THEN
			pEffectiveCtrl^.PackMLIn.eCommand := E_PackMLCommand.None;
			pEffectiveCtrl^.PackMLIn.bCommandChangeRequest := FALSE;
		END_IF
		
		// If an upper request is already high while control is unavailable, require it
		// to return low before it may be forwarded after the Module re-enters Execute.
		IF bUpperCommandHigh THEN _Entries[nIndex].UpperCommandBlockedUntilFalse := TRUE; END_IF
		IF bUpperModeHigh THEN _Entries[nIndex].UpperModeBlockedUntilFalse := TRUE; END_IF
		_Entries[nIndex].UpperCommandWasHigh := bUpperCommandHigh;
		_Entries[nIndex].UpperModeWasHigh := bUpperModeHigh;
		CONTINUE;
	END_IF
	
	// A low level re-arms the corresponding upper request channel.
	IF NOT bUpperCommandHigh THEN _Entries[nIndex].UpperCommandBlockedUntilFalse := FALSE; END_IF
	IF NOT bUpperModeHigh THEN _Entries[nIndex].UpperModeBlockedUntilFalse := FALSE; END_IF
	
	// A Service owned by a Composite accepts only the owner's internal command path;
	// direct upper commands and all upper mode changes remain suppressed.
	IF _Entries[nIndex].CompositeOwnerServiceId <> 0 THEN
		IF bUpperCommandHigh THEN _Entries[nIndex].UpperCommandBlockedUntilFalse := TRUE; END_IF
		IF bUpperModeHigh THEN _Entries[nIndex].UpperModeBlockedUntilFalse := TRUE; END_IF
		pEffectiveCtrl^.PackMLIn.eMode := E_PackMLMode.Unknown;
		pEffectiveCtrl^.PackMLIn.bModeChangeRequest := FALSE;
		
		// After acceptance or rejection, force one low scan to complete the request handshake.
		IF _Entries[nIndex].InternalRequestMustGoLow THEN
			pEffectiveCtrl^.PackMLIn.eCommand := E_PackMLCommand.None;
			pEffectiveCtrl^.PackMLIn.bCommandChangeRequest := FALSE;
			_Entries[nIndex].InternalRequestMustGoLow := FALSE;
			
		// Promote a queued command to the asserted request state, then hold it high
		// until M_ObserveCycle sees the matching Service response.
		ELSIF _Entries[nIndex].InternalCommandState = E_ServiceInternalCommandState.Queued THEN
			pEffectiveCtrl^.RequestId := _Entries[nIndex].InternalRequestId;
			pEffectiveCtrl^.PackMLIn.eCommand := _Entries[nIndex].InternalCommand;
			pEffectiveCtrl^.PackMLIn.bCommandChangeRequest := TRUE;
			_Entries[nIndex].InternalCommandState := E_ServiceInternalCommandState.RequestHigh;
			
		ELSIF _Entries[nIndex].InternalCommandState = E_ServiceInternalCommandState.RequestHigh THEN
			pEffectiveCtrl^.RequestId := _Entries[nIndex].InternalRequestId;
			pEffectiveCtrl^.PackMLIn.eCommand := _Entries[nIndex].InternalCommand;
			pEffectiveCtrl^.PackMLIn.bCommandChangeRequest := TRUE;
			
		ELSE
			pEffectiveCtrl^.PackMLIn.eCommand := E_PackMLCommand.None;
			pEffectiveCtrl^.PackMLIn.bCommandChangeRequest := FALSE;
		END_IF
		
		_Entries[nIndex].UpperCommandWasHigh := bUpperCommandHigh;
		_Entries[nIndex].UpperModeWasHigh := bUpperModeHigh;
		CONTINUE;
	END_IF
	
	// With no Composite owner, the Service normally follows its direct upper control.
	pEffectiveCtrl^ := pUpperCtrl^;
	IF _Entries[nIndex].UpperCommandBlockedUntilFalse THEN
		pEffectiveCtrl^.PackMLIn.bCommandChangeRequest := FALSE;
		
	ELSE
		// Snapshot parameters only on a newly asserted Start request. This keeps one
		// execution's effective parameters stable while the upper input remains high.
		bNewStartRequest := bUpperCommandHigh AND NOT _Entries[nIndex].UpperCommandWasHigh
			AND (pUpperCtrl^.PackMLIn.eCommand = E_PackMLCommand.Start);
		IF bNewStartRequest THEN
			MEMCPY(destAddr := _Entries[nIndex].EffectiveParamAddress,
				srcAddr := _Entries[nIndex].UpperParamAddress, n := _Entries[nIndex].ParameterSize);
		END_IF
	END_IF
	
	// Mode requests use the same return-low re-arm rule as command requests.
	IF _Entries[nIndex].UpperModeBlockedUntilFalse THEN
		pEffectiveCtrl^.PackMLIn.bModeChangeRequest := FALSE;
	END_IF
	
	_Entries[nIndex].UpperCommandWasHigh := bUpperCommandHigh;
	_Entries[nIndex].UpperModeWasHigh := bUpperModeHigh;
END_FOR
END_METHOD

METHOD PRIVATE M_ProcessOwnershipRequests
VAR
	nOrder : UINT;
	nIndex : UINT;
	nCandidateIndex : UINT;
	nDependency : UINT;
	nDependencyIndex : UINT;
	nLastServiceId : UDINT;
	nCandidateServiceId : UDINT;
	pDependencies : POINTER TO UDINT;
	bConflict : BOOL;
	bNotIdle : BOOL;
	bUnsupported : BOOL;
END_VAR
nLastServiceId := 0;
FOR nOrder := 1 TO _RegisteredCount DO
	nCandidateIndex := 0;
	nCandidateServiceId := 0;
	FOR nIndex := 1 TO _RegisteredCount DO
		IF (_Entries[nIndex].OwnershipState = E_CompositeOwnershipState.Pending)
			AND (_Entries[nIndex].ServiceId > nLastServiceId)
			AND ((nCandidateIndex = 0) OR (_Entries[nIndex].ServiceId < nCandidateServiceId)) THEN
			nCandidateIndex := nIndex;
			nCandidateServiceId := _Entries[nIndex].ServiceId;
		END_IF
	END_FOR
	IF nCandidateIndex = 0 THEN EXIT; END_IF
	nLastServiceId := nCandidateServiceId;
	bConflict := FALSE;
	bNotIdle := FALSE;
	bUnsupported := FALSE;
	pDependencies := _Entries[nCandidateIndex].CompositeDependenciesAddress;
	FOR nDependency := 1 TO _Entries[nCandidateIndex].CompositeDependencyCount DO
		nDependencyIndex := M_FindIndexByServiceId(ServiceId := pDependencies[nDependency - 1]);
		IF _Entries[nDependencyIndex].CompositeOwnerServiceId <> 0 THEN
			bConflict := TRUE;
		ELSIF NOT _Entries[nDependencyIndex].ObservedSnapshot.Valid
			OR (_Entries[nDependencyIndex].ObservedSnapshot.PackMLOut.eStateCurrent <> E_PackMLState.Idle) THEN
			bNotIdle := TRUE;
		ELSIF _Entries[nDependencyIndex].ObservedSnapshot.CompletionBehavior
			<> E_ServiceCompletionBehavior.NaturalCompletion THEN
			bUnsupported := TRUE;
		END_IF
	END_FOR
	IF bConflict THEN
		_Entries[nCandidateIndex].OwnershipState := E_CompositeOwnershipState.RejectedConflict;
	ELSIF bUnsupported THEN
		_Entries[nCandidateIndex].OwnershipState := E_CompositeOwnershipState.RejectedUnsupportedCompletionBehavior;
	ELSIF bNotIdle THEN
		_Entries[nCandidateIndex].OwnershipState := E_CompositeOwnershipState.RejectedDependencyNotIdle;
	ELSE
		FOR nDependency := 1 TO _Entries[nCandidateIndex].CompositeDependencyCount DO
			nDependencyIndex := M_FindIndexByServiceId(ServiceId := pDependencies[nDependency - 1]);
			_Entries[nDependencyIndex].CompositeOwnerServiceId := _Entries[nCandidateIndex].ServiceId;
		END_FOR
		_Entries[nCandidateIndex].OwnershipState := E_CompositeOwnershipState.Owned;
	END_IF
END_FOR
END_METHOD

METHOD PUBLIC FINAL M_Register : BOOL
VAR_INPUT
	ServiceId : UDINT;
	AllowCompositeCall : BOOL;
	UpperParam : ANY;
	EffectiveParam : ANY;
END_VAR
VAR_IN_OUT
	UpperCtrl : ST_ServiceCtrl;
	EffectiveCtrl : ST_ServiceCtrl;
	Status : ST_ServiceStatus;
END_VAR
VAR
	nIndex : UINT;
	nTargetIndex : UINT;
	nUpperParamSize : UDINT;
	nEffectiveParamSize : UDINT;
	sUpperParamType : STRING(255);
	sEffectiveParamType : STRING(255);
	hrUpperParam : HRESULT;
	hrEffectiveParam : HRESULT;
END_VAR
// 在 M_BeginRegistration 與 M_Seal 之間登錄一個 Service 的控制、參數與狀態儲存位置。
// 此方法保存呼叫端變數的位址而非內容，因此這些變數必須與 Coordinator 具有相同或更長生命週期。
M_Register := FALSE;
IF (_RegistrationError <> E_ServiceRegistrationError.None) OR NOT _RegistrationStarted THEN RETURN; END_IF

// 註冊封存後不可再新增；註冊錯誤採 first-error-wins，後續呼叫只會回傳 FALSE。
IF _Sealed THEN
	M_SetRegistrationError(Error := E_ServiceRegistrationError.RegistryAlreadySealed, ServiceId := ServiceId);
	RETURN;
END_IF
IF ServiceId = 0 THEN
	M_SetRegistrationError(Error := E_ServiceRegistrationError.InvalidServiceId, ServiceId := ServiceId);
	RETURN;
END_IF
FOR nIndex := 1 TO _RegisteredCount DO
	IF _Entries[nIndex].ServiceId = ServiceId THEN
		M_SetRegistrationError(Error := E_ServiceRegistrationError.DuplicateServiceId, ServiceId := ServiceId);
		RETURN;
	END_IF
END_FOR
IF _RegisteredCount >= Param_Config.MaxServicesPerModule THEN
	M_SetRegistrationError(Error := E_ServiceRegistrationError.CapacityExceeded, ServiceId := ServiceId);
	RETURN;
END_IF

// 控制、狀態與 ANY 參數都必須指向有效儲存空間。
IF (ADR(UpperCtrl) = 0) OR (ADR(EffectiveCtrl) = 0) OR (ADR(Status) = 0)
	OR (UpperParam.pValue = 0) OR (EffectiveParam.pValue = 0)
	OR (UpperParam.diSize <= 0) OR (EffectiveParam.diSize <= 0) THEN
	M_SetRegistrationError(Error := E_ServiceRegistrationError.InvalidStorage, ServiceId := ServiceId);
	RETURN;
END_IF
nUpperParamSize := DINT_TO_UDINT(UpperParam.diSize);
nEffectiveParamSize := DINT_TO_UDINT(EffectiveParam.diSize);

// Upper 與 Effective 參數不只大小必須相同，實際 DUT 型別名稱也必須一致。
IF nUpperParamSize <> nEffectiveParamSize THEN
	M_SetRegistrationError(Error := E_ServiceRegistrationError.ParameterSizeMismatch, ServiceId := ServiceId);
	RETURN;
END_IF
sUpperParamType := _JsonDataType.GetDataTypeNameByAddress(
	nData := nUpperParamSize, pData := UpperParam.pValue, hrErrorCode => hrUpperParam);
sEffectiveParamType := _JsonDataType.GetDataTypeNameByAddress(
	nData := nEffectiveParamSize, pData := EffectiveParam.pValue, hrErrorCode => hrEffectiveParam);
IF (hrUpperParam <> 0) OR (hrEffectiveParam <> 0) OR (sUpperParamType = '') OR (sEffectiveParamType = '') THEN
	M_SetRegistrationError(Error := E_ServiceRegistrationError.ParameterTypeResolutionFailed, ServiceId := ServiceId);
	RETURN;
END_IF
IF sUpperParamType <> sEffectiveParamType THEN
	M_SetRegistrationError(Error := E_ServiceRegistrationError.ParameterTypeMismatch, ServiceId := ServiceId);
	RETURN;
END_IF

// 所有驗證通過後才提交 entry，避免留下半完成的註冊資料。
nTargetIndex := _RegisteredCount + 1;
_Entries[nTargetIndex].InUse := TRUE;
_Entries[nTargetIndex].ServiceId := ServiceId;
_Entries[nTargetIndex].AllowCompositeCall := AllowCompositeCall;
_Entries[nTargetIndex].UpperCtrlAddress := ADR(UpperCtrl);
_Entries[nTargetIndex].EffectiveCtrlAddress := ADR(EffectiveCtrl);
_Entries[nTargetIndex].UpperParamAddress := UpperParam.pValue;
_Entries[nTargetIndex].EffectiveParamAddress := EffectiveParam.pValue;
_Entries[nTargetIndex].ParameterSize := nUpperParamSize;
_Entries[nTargetIndex].ParameterTypeName := sUpperParamType;
_Entries[nTargetIndex].StatusAddress := ADR(Status);
_Entries[nTargetIndex].InternalCommandState := E_ServiceInternalCommandState.None;
_Entries[nTargetIndex].OwnershipState := E_CompositeOwnershipState.None;
_RegisteredCount := nTargetIndex;
M_Register := TRUE;
END_METHOD

METHOD PUBLIC FINAL M_RegisterCompositeDefinition : BOOL
VAR_INPUT
	CompositeServiceId : UDINT;
	DependencyCount : UINT;
END_VAR
VAR_IN_OUT
	DependencyIds : ARRAY[1..Param_Config.MaxCompositeDependencies] OF UDINT;
END_VAR
VAR
	nCompositeIndex : UINT;
	nDependencyIndex : UINT;
	nDependency : UINT;
	nOtherDependency : UINT;
END_VAR
// 為已註冊的 Composite Service 宣告可呼叫的 dependency 清單；應在所有 Service 註冊後、M_Seal 前呼叫。
// DependencyIds 的位址會被保存而非複製，因此陣列必須在 Coordinator 使用期間持續存在且不得任意改寫。
M_RegisterCompositeDefinition := FALSE;
IF (_RegistrationError <> E_ServiceRegistrationError.None) OR NOT _RegistrationStarted THEN RETURN; END_IF
IF _Sealed THEN
	M_SetRegistrationError(Error := E_ServiceRegistrationError.RegistryAlreadySealed, ServiceId := CompositeServiceId);
	RETURN;
END_IF
nCompositeIndex := M_FindIndexByServiceId(ServiceId := CompositeServiceId);
IF nCompositeIndex = 0 THEN
	M_SetRegistrationError(Error := E_ServiceRegistrationError.InvalidCompositeService, ServiceId := CompositeServiceId);
	RETURN;
END_IF
IF _Entries[nCompositeIndex].IsComposite THEN
	M_SetRegistrationError(Error := E_ServiceRegistrationError.DuplicateCompositeDefinition, ServiceId := CompositeServiceId);
	RETURN;
END_IF
IF DependencyCount = 0 THEN
	M_SetRegistrationError(Error := E_ServiceRegistrationError.EmptyCompositeDependencyList, ServiceId := CompositeServiceId);
	RETURN;
END_IF
IF DependencyCount > Param_Config.MaxCompositeDependencies THEN
	M_SetRegistrationError(Error := E_ServiceRegistrationError.CompositeDependencyCapacityExceeded, ServiceId := CompositeServiceId);
	RETURN;
END_IF

// 每個 dependency 必須已註冊、允許 Composite 呼叫，且不可指向自己或在清單中重複。
FOR nDependency := 1 TO DependencyCount DO
	IF DependencyIds[nDependency] = 0 THEN
		M_SetRegistrationError(Error := E_ServiceRegistrationError.InvalidCompositeDependencyId, ServiceId := CompositeServiceId);
		RETURN;
	END_IF
	IF DependencyIds[nDependency] = CompositeServiceId THEN
		M_SetRegistrationError(Error := E_ServiceRegistrationError.SelfDependency, ServiceId := CompositeServiceId);
		RETURN;
	END_IF
	nDependencyIndex := M_FindIndexByServiceId(ServiceId := DependencyIds[nDependency]);
	IF nDependencyIndex = 0 THEN
		M_SetRegistrationError(Error := E_ServiceRegistrationError.UnknownCompositeDependency, ServiceId := DependencyIds[nDependency]);
		RETURN;
	END_IF
	IF NOT _Entries[nDependencyIndex].AllowCompositeCall THEN
		M_SetRegistrationError(Error := E_ServiceRegistrationError.CompositeDependencyNotAllowed, ServiceId := DependencyIds[nDependency]);
		RETURN;
	END_IF
	FOR nOtherDependency := 1 TO nDependency - 1 DO
		IF DependencyIds[nOtherDependency] = DependencyIds[nDependency] THEN
			M_SetRegistrationError(Error := E_ServiceRegistrationError.DuplicateCompositeDependency, ServiceId := DependencyIds[nDependency]);
			RETURN;
		END_IF
	END_FOR
END_FOR

// 驗證完成後一次提交 definition；nested Composite 會在 M_Seal 統一拒絕。
_Entries[nCompositeIndex].IsComposite := TRUE;
_Entries[nCompositeIndex].CompositeDependenciesAddress := ADR(DependencyIds);
_Entries[nCompositeIndex].CompositeDependencyCount := DependencyCount;
_Entries[nCompositeIndex].OwnershipState := E_CompositeOwnershipState.None;
M_RegisterCompositeDefinition := TRUE;
END_METHOD

METHOD PUBLIC FINAL M_ReleaseCompositeOwnership : BOOL
VAR_INPUT
	CompositeServiceId : UDINT;
END_VAR
VAR
	nCompositeIndex : UINT;
	nDependencyIndex : UINT;
	nDependency : UINT;
	pDependencies : POINTER TO UDINT;
	pEffectiveCtrl : POINTER TO ST_ServiceCtrl;
END_VAR
// 釋放 Composite 實際持有的所有 dependency；未知或非 Composite Service 會回傳 FALSE。
// 通常在 sequence 完成、Stop、Abort、Clear 或 Reset 清理階段呼叫。
M_ReleaseCompositeOwnership := FALSE;
nCompositeIndex := M_FindIndexByServiceId(ServiceId := CompositeServiceId);
IF (nCompositeIndex = 0) OR NOT _Entries[nCompositeIndex].IsComposite THEN RETURN; END_IF
pDependencies := _Entries[nCompositeIndex].CompositeDependenciesAddress;
FOR nDependency := 1 TO _Entries[nCompositeIndex].CompositeDependencyCount DO
	nDependencyIndex := M_FindIndexByServiceId(ServiceId := pDependencies[nDependency - 1]);

	// 只清除仍屬於此 Composite 的 dependency，避免破壞其他 owner 後續取得的 ownership。
	IF _Entries[nDependencyIndex].CompositeOwnerServiceId = CompositeServiceId THEN
		_Entries[nDependencyIndex].CompositeOwnerServiceId := 0;

		// 尚未完成的內部命令標記為 Cancelled，並立即撤除送往 Service 的 request high。
		IF (_Entries[nDependencyIndex].InternalCommandState = E_ServiceInternalCommandState.Queued)
			OR (_Entries[nDependencyIndex].InternalCommandState = E_ServiceInternalCommandState.RequestHigh) THEN
			_Entries[nDependencyIndex].InternalCommandState := E_ServiceInternalCommandState.Cancelled;
		END_IF
		_Entries[nDependencyIndex].InternalRequestMustGoLow := FALSE;
		pEffectiveCtrl := _Entries[nDependencyIndex].EffectiveCtrlAddress;
		pEffectiveCtrl^.PackMLIn.bCommandChangeRequest := FALSE;
	END_IF
END_FOR

// Composite 回到 None；下次使用前必須重新呼叫 M_RequestCompositeOwnership。
_Entries[nCompositeIndex].OwnershipState := E_CompositeOwnershipState.None;
M_ReleaseCompositeOwnership := TRUE;
END_METHOD

METHOD PUBLIC FINAL M_RequestCompositeOwnership : BOOL
VAR_INPUT
	CompositeServiceId : UDINT;
END_VAR
VAR
	nIndex : UINT;
END_VAR
// 提出取得 Composite 全部 dependency ownership 的請求；Coordinator 必須已完成註冊並 Ready。
// 回傳 TRUE 只代表請求已接受或原本已持有，不代表本次呼叫已立即取得 ownership。
M_RequestCompositeOwnership := FALSE;
IF NOT Ready THEN RETURN; END_IF
nIndex := M_FindIndexByServiceId(ServiceId := CompositeServiceId);
IF (nIndex = 0) OR NOT _Entries[nIndex].IsComposite THEN RETURN; END_IF

// 已持有時採 idempotent 成功；其他狀態則重新排入 Pending。
IF _Entries[nIndex].OwnershipState = E_CompositeOwnershipState.Owned THEN
	M_RequestCompositeOwnership := TRUE;
	RETURN;
END_IF

// M_PrepareCycle 會在 Module Execute 期間以原子方式解析 Pending，結果需另行查詢。
_Entries[nIndex].OwnershipState := E_CompositeOwnershipState.Pending;
M_RequestCompositeOwnership := TRUE;
END_METHOD

METHOD PUBLIC FINAL M_Seal : BOOL
VAR
	nIndex : UINT;
	nDependency : UINT;
	nDependencyIndex : UINT;
	pDependencies : POINTER TO UDINT;
	pEffectiveCtrl : POINTER TO ST_ServiceCtrl;
END_VAR
// 結束一次性註冊階段並使 Ready 成立；所有 Service 與 Composite definition 都必須先完成。
// 封存失敗會留下穩定的 RegistrationError，且 registry 不會進入可執行狀態。
M_Seal := FALSE;
IF _RegistrationError <> E_ServiceRegistrationError.None THEN RETURN; END_IF

IF _Sealed THEN
	M_SetRegistrationError(Error := E_ServiceRegistrationError.RegistryAlreadySealed, ServiceId := 0);
	RETURN;
END_IF

IF NOT _RegistrationStarted OR (_RegisteredCount = 0) THEN
	M_SetRegistrationError(Error := E_ServiceRegistrationError.EmptyRegistry, ServiceId := 0);
	RETURN;
END_IF

// Composite 不可依賴另一個 Composite，避免形成巢狀 ownership 與不明確的控制優先序。
FOR nIndex := 1 TO _RegisteredCount DO
	IF _Entries[nIndex].IsComposite THEN
		pDependencies := _Entries[nIndex].CompositeDependenciesAddress;
		FOR nDependency := 1 TO _Entries[nIndex].CompositeDependencyCount DO
			nDependencyIndex := M_FindIndexByServiceId(ServiceId := pDependencies[nDependency - 1]);
			IF _Entries[nDependencyIndex].IsComposite THEN
				M_SetRegistrationError(Error := E_ServiceRegistrationError.NestedCompositeNotSupported,
					ServiceId := _Entries[nDependencyIndex].ServiceId);
				RETURN;
			END_IF
		END_FOR
	END_IF
END_FOR

// 封存時將所有有效控制 request 拉低並清除舊快照，建立一致的首個執行週期。
FOR nIndex := 1 TO _RegisteredCount DO
	pEffectiveCtrl := _Entries[nIndex].EffectiveCtrlAddress;
	pEffectiveCtrl^.PackMLIn.bCommandChangeRequest := FALSE;
	pEffectiveCtrl^.PackMLIn.bModeChangeRequest := FALSE;
	_Entries[nIndex].ObservedSnapshot.Valid := FALSE;
END_FOR
_AllIdle := FALSE;
_AllStopped := FALSE;
_AllAborted := FALSE;

// _Sealed 最後才設為 TRUE，確保 Ready 不會看見部分初始化的 registry。
_Sealed := TRUE;
M_Seal := TRUE;
END_METHOD

METHOD PRIVATE M_SetRegistrationError
VAR_INPUT
	Error : E_ServiceRegistrationError;
	ServiceId : UDINT;
END_VAR
IF _RegistrationError <> E_ServiceRegistrationError.None THEN RETURN; END_IF
_RegistrationError := Error;
_FailedServiceId := ServiceId;
_Sealed := FALSE;
_AllIdle := FALSE;
_AllStopped := FALSE;
_AllAborted := FALSE;
END_METHOD

METHOD PUBLIC FINAL M_SubmitInternalCommand : E_ServiceCallSubmitResult
VAR_INPUT
	CallerServiceId : UDINT;
	TargetServiceId : UDINT;
	RequestId : UDINT;
	Command : E_PackMLCommand;
END_VAR
VAR
	nCallerIndex : UINT;
	nTargetIndex : UINT;
END_VAR
// 由 Composite owner 對 dependency 排入 lifecycle 命令（Stop、Abort、Clear、Reset）。
// 方法只負責驗證與 queue；M_PrepareCycle 才會輸出 request，M_ObserveCycle 再判讀回覆。
IF NOT Ready THEN
	M_SubmitInternalCommand := E_ServiceCallSubmitResult.CoordinatorNotReady;
	RETURN;
END_IF

// Start 必須使用 M_SubmitInternalStart，以便在送出命令前驗證並快照參數。
IF (Command <> E_PackMLCommand.Stop) AND (Command <> E_PackMLCommand.Abort)
	AND (Command <> E_PackMLCommand.Clear) AND (Command <> E_PackMLCommand.Reset) THEN
	M_SubmitInternalCommand := E_ServiceCallSubmitResult.InvalidCommand;
	RETURN;
END_IF

nTargetIndex := M_FindIndexByServiceId(ServiceId := TargetServiceId);
IF nTargetIndex = 0 THEN
	M_SubmitInternalCommand := E_ServiceCallSubmitResult.UnknownService;
	RETURN;
END_IF

nCallerIndex := M_FindIndexByServiceId(ServiceId := CallerServiceId);

// Caller 必須是有宣告此 Target 的 Composite，且目前確實持有該 dependency。
IF (nCallerIndex = 0) OR NOT M_IsDeclaredDependency(
	CompositeIndex := nCallerIndex, TargetServiceId := TargetServiceId) THEN
	M_SubmitInternalCommand := E_ServiceCallSubmitResult.DependencyNotDeclared;
	RETURN;
END_IF
IF _Entries[nTargetIndex].CompositeOwnerServiceId <> CallerServiceId THEN
	M_SubmitInternalCommand := E_ServiceCallSubmitResult.NotOwner;
	RETURN;
END_IF

// 一個 Target 同時間只允許一筆內部請求；包含等待強制 low 的 scan 都視為 Busy。
IF (_Entries[nTargetIndex].InternalCommandState = E_ServiceInternalCommandState.Queued)
	OR (_Entries[nTargetIndex].InternalCommandState = E_ServiceInternalCommandState.RequestHigh)
	OR _Entries[nTargetIndex].InternalRequestMustGoLow THEN
	M_SubmitInternalCommand := E_ServiceCallSubmitResult.Busy;
	RETURN;
END_IF

// 所有驗證通過後才提交 RequestId 與命令，供後續 response correlation 使用。
_Entries[nTargetIndex].InternalRequestId := RequestId;
_Entries[nTargetIndex].InternalCommand := Command;
_Entries[nTargetIndex].InternalCommandState := E_ServiceInternalCommandState.Queued;
_Entries[nTargetIndex].InternalRequestMustGoLow := FALSE;
M_SubmitInternalCommand := E_ServiceCallSubmitResult.Queued;
END_METHOD

METHOD PUBLIC FINAL M_SubmitInternalStart : E_ServiceCallSubmitResult
VAR_INPUT
	CallerServiceId : UDINT;
	TargetServiceId : UDINT;
	RequestId : UDINT;
	Parameters : ANY;
END_VAR
VAR
	nCallerIndex : UINT;
	nTargetIndex : UINT;
	nParameterSize : UDINT;
	sParameterType : STRING(255);
	hrParameter : HRESULT;
END_VAR
// 由 Composite owner 對 dependency 排入 Start，並在排入當下快照本次執行參數。
// 方法只負責驗證、複製與 queue；實際 request high 由 M_PrepareCycle 在後續週期輸出。
IF NOT Ready THEN
	M_SubmitInternalStart := E_ServiceCallSubmitResult.CoordinatorNotReady;
	RETURN;
END_IF
nTargetIndex := M_FindIndexByServiceId(ServiceId := TargetServiceId);
IF nTargetIndex = 0 THEN
	M_SubmitInternalStart := E_ServiceCallSubmitResult.UnknownService;
	RETURN;
END_IF
nCallerIndex := M_FindIndexByServiceId(ServiceId := CallerServiceId);

// Caller 必須宣告 Target 為 dependency，並先成功取得該 Target 的 ownership。
IF (nCallerIndex = 0) OR NOT M_IsDeclaredDependency(
	CompositeIndex := nCallerIndex, TargetServiceId := TargetServiceId) THEN
	M_SubmitInternalStart := E_ServiceCallSubmitResult.DependencyNotDeclared;
	RETURN;
END_IF
IF _Entries[nTargetIndex].CompositeOwnerServiceId <> CallerServiceId THEN
	M_SubmitInternalStart := E_ServiceCallSubmitResult.NotOwner;
	RETURN;
END_IF

// 前一筆請求尚在 queue、維持 high 或等待 low 時，不可覆寫參數與 RequestId。
IF (_Entries[nTargetIndex].InternalCommandState = E_ServiceInternalCommandState.Queued)
	OR (_Entries[nTargetIndex].InternalCommandState = E_ServiceInternalCommandState.RequestHigh)
	OR _Entries[nTargetIndex].InternalRequestMustGoLow THEN
	M_SubmitInternalStart := E_ServiceCallSubmitResult.Busy;
	RETURN;
END_IF
IF (Parameters.pValue = 0) OR (Parameters.diSize <= 0) THEN
	M_SubmitInternalStart := E_ServiceCallSubmitResult.ParameterSizeMismatch;
	RETURN;
END_IF

// ANY 參數的大小與實際 DUT 型別都必須和 M_Register 記錄的 Target 參數一致。
nParameterSize := DINT_TO_UDINT(Parameters.diSize);
IF nParameterSize <> _Entries[nTargetIndex].ParameterSize THEN
	M_SubmitInternalStart := E_ServiceCallSubmitResult.ParameterSizeMismatch;
	RETURN;
END_IF
sParameterType := _JsonDataType.GetDataTypeNameByAddress(
	nData := nParameterSize, pData := Parameters.pValue, hrErrorCode => hrParameter);
IF (hrParameter <> 0) OR (sParameterType = '') THEN
	M_SubmitInternalStart := E_ServiceCallSubmitResult.ParameterTypeResolutionFailed;
	RETURN;
END_IF
IF sParameterType <> _Entries[nTargetIndex].ParameterTypeName THEN
	M_SubmitInternalStart := E_ServiceCallSubmitResult.ParameterTypeMismatch;
	RETURN;
END_IF

// 驗證完成後先複製參數，再提交 Start request，確保 Service 不會看到半更新資料。
MEMCPY(destAddr := _Entries[nTargetIndex].EffectiveParamAddress,
	srcAddr := Parameters.pValue, n := nParameterSize);
_Entries[nTargetIndex].InternalRequestId := RequestId;
_Entries[nTargetIndex].InternalCommand := E_PackMLCommand.Start;
_Entries[nTargetIndex].InternalCommandState := E_ServiceInternalCommandState.Queued;
_Entries[nTargetIndex].InternalRequestMustGoLow := FALSE;
M_SubmitInternalStart := E_ServiceCallSubmitResult.Queued;
END_METHOD

PROPERTY PUBLIC FINAL Ready : BOOL
GET
Ready := _RegistrationStarted AND _Sealed
	AND (_RegistrationError = E_ServiceRegistrationError.None);
END_GET
END_PROPERTY

PROPERTY PUBLIC FINAL RegisteredCount : UINT
GET
RegisteredCount := _RegisteredCount;
END_GET
END_PROPERTY

PROPERTY PUBLIC FINAL RegistrationError : E_ServiceRegistrationError
GET
RegistrationError := _RegistrationError;
END_GET
END_PROPERTY

END_FUNCTION_BLOCK

// ---- POUs/20_Service/FB_CompositeServiceBase.TcPOU
FUNCTION_BLOCK FB_CompositeServiceBase EXTENDS FB_ServiceBase
VAR
	_Coordinator : REFERENCE TO FB_ServiceCoordinator;
	_ServiceCaller : FB_ServiceCaller;
	_DependencyServiceIds : ARRAY[1..Param_Config.MaxCompositeDependencies] OF UDINT;
	_DependencyCount : UINT;
	_Configured : BOOL;
	_DefinitionAttempted : BOOL;
	_DefinitionOpen : BOOL;
	_DependencyOverflow : BOOL;
	_OwnershipRequested : BOOL;
	_OwnershipHeld : BOOL;
	_SequenceFailed : BOOL;
	_LifecycleCommandSubmitted : ARRAY[1..Param_Config.MaxCompositeDependencies] OF BOOL;
END_VAR

METHOD PROTECTED H_DeclareServices
// Derived Composite Services declare dependencies through M_AddDependency().
END_METHOD

METHOD PROTECTED FINAL H_OnAborting : E_PackMLHookResult
VAR_INPUT
	bFirstScan : BOOL;
END_VAR
VAR
	nDependency : UINT;
	bAllSafe : BOOL;
	Snapshot : ST_ServiceExecutionSnapshot;
END_VAR
H_OnAborting := E_PackMLHookResult.Busy;
IF bFirstScan THEN M_ClearLifecycleRequests(); END_IF
IF NOT _OwnershipHeld THEN
	H_OnAborting := E_PackMLHookResult.Done;
	RETURN;
END_IF
bAllSafe := TRUE;
FOR nDependency := 1 TO _DependencyCount DO
	IF NOT M_GetDependencySnapshot(DependencyIndex := nDependency, Snapshot => Snapshot) THEN
		bAllSafe := FALSE;
		CONTINUE;
	END_IF
	CASE Snapshot.PackMLOut.eStateCurrent OF
		E_PackMLState.Idle, E_PackMLState.Stopped, E_PackMLState.Aborted:
			;
	ELSE
		bAllSafe := FALSE;
		M_EnsureLifecycleCommand(DependencyIndex := nDependency, Command := E_PackMLCommand.Abort);
	END_CASE
END_FOR
IF bAllSafe THEN H_OnAborting := E_PackMLHookResult.Done; END_IF
END_METHOD

METHOD PROTECTED FINAL H_OnClearing : E_PackMLHookResult
VAR_INPUT
	bFirstScan : BOOL;
END_VAR
VAR
	nDependency : UINT;
	bAllSafe : BOOL;
	Snapshot : ST_ServiceExecutionSnapshot;
END_VAR
H_OnClearing := E_PackMLHookResult.Busy;

IF bFirstScan THEN M_ClearLifecycleRequests(); END_IF
IF NOT _OwnershipHeld THEN
	M_ClearAllError();
	H_OnClearing := E_PackMLHookResult.Done;
	RETURN;
END_IF

bAllSafe := TRUE;
FOR nDependency := 1 TO _DependencyCount DO
	IF NOT M_GetDependencySnapshot(DependencyIndex := nDependency, Snapshot => Snapshot) THEN
		bAllSafe := FALSE;
		CONTINUE;
	END_IF
	CASE Snapshot.PackMLOut.eStateCurrent OF
		E_PackMLState.Idle, E_PackMLState.Stopped:
			;
		E_PackMLState.Aborted:
			bAllSafe := FALSE;
			M_EnsureLifecycleCommand(DependencyIndex := nDependency, Command := E_PackMLCommand.Clear);
	ELSE
		bAllSafe := FALSE;
	END_CASE
END_FOR

IF bAllSafe THEN
	M_ClearAllError();
	H_OnClearing := E_PackMLHookResult.Done;
END_IF
END_METHOD

METHOD PROTECTED FINAL H_OnComplete
VAR_INPUT
	bFirstScan : BOOL;
END_VAR
// Normal completion releases ownership in H_OnCompleting.
END_METHOD

METHOD PROTECTED FINAL H_OnCompleting : E_PackMLHookResult
VAR_INPUT
	bFirstScan : BOOL;
END_VAR
VAR
	nDependency : UINT;
	bAllIdle : BOOL;
	Snapshot : ST_ServiceExecutionSnapshot;
END_VAR
H_OnCompleting := E_PackMLHookResult.Busy;
IF bFirstScan THEN M_ClearLifecycleRequests(); END_IF
IF NOT _OwnershipHeld THEN
	H_OnCompleting := E_PackMLHookResult.Done;
	RETURN;
END_IF
bAllIdle := TRUE;
FOR nDependency := 1 TO _DependencyCount DO
	IF NOT M_GetDependencySnapshot(DependencyIndex := nDependency, Snapshot => Snapshot) THEN
		bAllIdle := FALSE;
		CONTINUE;
	END_IF
	CASE Snapshot.PackMLOut.eStateCurrent OF
		E_PackMLState.Idle:
			;
		E_PackMLState.Complete:
			bAllIdle := FALSE;
			M_EnsureLifecycleCommand(DependencyIndex := nDependency, Command := E_PackMLCommand.Reset);
		E_PackMLState.Stopped:
			M_AddError(MainErrorId := TO_UDINT(E_CompositeServiceErrorCode.ChildStoppedUnexpectedly),
				SourceErrorId := TO_UDINT(Snapshot.PackMLOut.eStateErrorID),
				Message := 'A Composite dependency stopped while completing.');
			RequestCommand(eTargetCmd := E_PackMLCommand.Stop);
			RETURN;
		E_PackMLState.Aborted:
			M_AddError(MainErrorId := TO_UDINT(E_CompositeServiceErrorCode.ChildAbortedUnexpectedly),
				SourceErrorId := TO_UDINT(Snapshot.PackMLOut.eStateErrorID),
				Message := 'A Composite dependency aborted while completing.');
			RequestCommand(eTargetCmd := E_PackMLCommand.Abort);
			RETURN;
	ELSE
		bAllIdle := FALSE;
	END_CASE
END_FOR
IF bAllIdle THEN
	_Coordinator.M_ReleaseCompositeOwnership(CompositeServiceId := ServiceId);
	_OwnershipHeld := FALSE;
	_OwnershipRequested := FALSE;
	H_OnCompleting := E_PackMLHookResult.Done;
END_IF
END_METHOD

METHOD PROTECTED H_OnCompositeExecute : E_PackMLHookResult
VAR_INPUT
	bFirstScan : BOOL;
END_VAR
// Derived Composite Services implement their ordered process here.
H_OnCompositeExecute := E_PackMLHookResult.Busy;
END_METHOD

METHOD PROTECTED FINAL H_OnExecute : E_PackMLHookResult
VAR_INPUT
	bFirstScan : BOOL;
END_VAR
VAR
	nDependency : UINT;
	Snapshot : ST_ServiceExecutionSnapshot;
END_VAR
H_OnExecute := E_PackMLHookResult.Busy;
IF bFirstScan THEN _SequenceFailed := FALSE; END_IF
FOR nDependency := 1 TO _DependencyCount DO
	IF NOT M_GetDependencySnapshot(DependencyIndex := nDependency, Snapshot => Snapshot) THEN
		M_FailSequence(ErrorCode := E_CompositeServiceErrorCode.InvalidSequenceState,
			FailedServiceId := _DependencyServiceIds[nDependency], SourceErrorId := 0,
			Message := 'A Composite dependency snapshot is unavailable.');
		EXIT;
	END_IF
	IF Snapshot.PackMLOut.eStateCurrent = E_PackMLState.Aborted THEN
		M_AddError(MainErrorId := TO_UDINT(E_CompositeServiceErrorCode.ChildAbortedUnexpectedly),
			SourceErrorId := TO_UDINT(Snapshot.PackMLOut.eStateErrorID),
			Message := 'A Composite dependency aborted during Execute.');
		RequestCommand(eTargetCmd := E_PackMLCommand.Abort);
		RETURN;
	ELSIF Snapshot.PackMLOut.eStateCurrent = E_PackMLState.Stopped THEN
		M_AddError(MainErrorId := TO_UDINT(E_CompositeServiceErrorCode.ChildStoppedUnexpectedly),
			SourceErrorId := TO_UDINT(Snapshot.PackMLOut.eStateErrorID),
			Message := 'A Composite dependency stopped during Execute.');
		RequestCommand(eTargetCmd := E_PackMLCommand.Stop);
		RETURN;
	END_IF
END_FOR
IF NOT _SequenceFailed THEN
	H_OnExecute := H_OnCompositeExecute(bFirstScan := bFirstScan);
END_IF
IF _SequenceFailed THEN
	RequestCommand(eTargetCmd := E_PackMLCommand.Stop);
	H_OnExecute := E_PackMLHookResult.Busy;
END_IF
END_METHOD

METHOD PROTECTED FINAL H_OnIdle
VAR_INPUT
	bFirstScan : BOOL;
END_VAR
IF bFirstScan THEN
	_SequenceFailed := FALSE;
	IF _OwnershipHeld AND __ISVALIDREF(_Coordinator) THEN
		_Coordinator.M_ReleaseCompositeOwnership(CompositeServiceId := ServiceId);
		_OwnershipHeld := FALSE;
	END_IF
	_OwnershipRequested := FALSE;
END_IF
END_METHOD

METHOD PROTECTED FINAL H_OnResetting : E_PackMLHookResult
VAR_INPUT
	bFirstScan : BOOL;
END_VAR
VAR
	nDependency : UINT;
	bAllIdle : BOOL;
	Snapshot : ST_ServiceExecutionSnapshot;
END_VAR
H_OnResetting := E_PackMLHookResult.Busy;
IF bFirstScan THEN
	M_ClearLifecycleRequests();
	MEMSET(ADR(Status.ErrorList), 0, SIZEOF(Status.ErrorList));
END_IF
IF NOT _OwnershipHeld THEN
	H_OnResetting := E_PackMLHookResult.Done;
	RETURN;
END_IF
bAllIdle := TRUE;
FOR nDependency := 1 TO _DependencyCount DO
	IF NOT M_GetDependencySnapshot(DependencyIndex := nDependency, Snapshot => Snapshot) THEN
		bAllIdle := FALSE;
		CONTINUE;
	END_IF
	CASE Snapshot.PackMLOut.eStateCurrent OF
		E_PackMLState.Idle:
			;
		E_PackMLState.Stopped, E_PackMLState.Complete:
			bAllIdle := FALSE;
			M_EnsureLifecycleCommand(DependencyIndex := nDependency, Command := E_PackMLCommand.Reset);
		E_PackMLState.Aborted:
			bAllIdle := FALSE;
			M_AddError(MainErrorId := TO_UDINT(E_CompositeServiceErrorCode.ChildAbortedUnexpectedly),
				SourceErrorId := TO_UDINT(Snapshot.PackMLOut.eStateErrorID),
				Message := 'A Composite dependency aborted while resetting.');
			RequestCommand(eTargetCmd := E_PackMLCommand.Abort);
	ELSE
		bAllIdle := FALSE;
	END_CASE
END_FOR
IF bAllIdle THEN
	_Coordinator.M_ReleaseCompositeOwnership(CompositeServiceId := ServiceId);
	_OwnershipHeld := FALSE;
	_OwnershipRequested := FALSE;
	H_OnResetting := E_PackMLHookResult.Done;
END_IF
END_METHOD

METHOD PROTECTED FINAL H_OnStarting : E_PackMLHookResult
VAR_INPUT
	bFirstScan : BOOL;
END_VAR
VAR
	OwnershipState : E_CompositeOwnershipState;
END_VAR
H_OnStarting := E_PackMLHookResult.Busy;
IF NOT _Configured OR NOT __ISVALIDREF(_Coordinator) THEN
	M_AddError(MainErrorId := TO_UDINT(E_CompositeServiceErrorCode.NotConfigured), SourceErrorId := 0,
		Message := 'Composite Service definition is not configured.');
	RequestCommand(eTargetCmd := E_PackMLCommand.Stop);
	RETURN;
END_IF
IF bFirstScan THEN
	_SequenceFailed := FALSE;
	_OwnershipRequested := _Coordinator.M_RequestCompositeOwnership(CompositeServiceId := ServiceId);
	IF NOT _OwnershipRequested THEN
		M_AddError(MainErrorId := TO_UDINT(E_CompositeServiceErrorCode.NotConfigured), SourceErrorId := 0,
			Message := 'Composite ownership request could not be submitted.');
		RequestCommand(eTargetCmd := E_PackMLCommand.Stop);
		RETURN;
	END_IF
END_IF
OwnershipState := _Coordinator.M_GetCompositeOwnershipState(CompositeServiceId := ServiceId);
CASE OwnershipState OF
	E_CompositeOwnershipState.Pending:
		;
	E_CompositeOwnershipState.Owned:
		_OwnershipHeld := TRUE;
		H_OnStarting := E_PackMLHookResult.Done;
	E_CompositeOwnershipState.RejectedConflict:
		M_AddError(MainErrorId := TO_UDINT(E_CompositeServiceErrorCode.OwnershipConflict),
			SourceErrorId := TO_UDINT(OwnershipState), Message := 'A Composite dependency is owned by another Composite.');
		RequestCommand(eTargetCmd := E_PackMLCommand.Stop);
	E_CompositeOwnershipState.RejectedDependencyNotIdle:
		M_AddError(MainErrorId := TO_UDINT(E_CompositeServiceErrorCode.DependencyNotIdle),
			SourceErrorId := TO_UDINT(OwnershipState), Message := 'A Composite dependency is not Idle.');
		RequestCommand(eTargetCmd := E_PackMLCommand.Stop);
	E_CompositeOwnershipState.RejectedUnsupportedCompletionBehavior:
		M_AddError(MainErrorId := TO_UDINT(E_CompositeServiceErrorCode.UnsupportedCompletionBehavior),
			SourceErrorId := TO_UDINT(OwnershipState), Message := 'A Composite dependency is not NaturalCompletion.');
		RequestCommand(eTargetCmd := E_PackMLCommand.Stop);
	E_CompositeOwnershipState.Cancelled:
		RequestCommand(eTargetCmd := E_PackMLCommand.Stop);
ELSE
	IF _OwnershipRequested THEN
		M_AddError(MainErrorId := TO_UDINT(E_CompositeServiceErrorCode.NotConfigured), SourceErrorId := 0,
			Message := 'Composite ownership state is unavailable.');
		RequestCommand(eTargetCmd := E_PackMLCommand.Stop);
	END_IF
END_CASE
END_METHOD

METHOD PROTECTED FINAL H_OnStopped
VAR_INPUT
	bFirstScan : BOOL;
END_VAR
// Ownership is intentionally retained until Reset returns every dependency to Idle.
END_METHOD

METHOD PROTECTED FINAL H_OnStopping : E_PackMLHookResult
VAR_INPUT
	bFirstScan : BOOL;
END_VAR
VAR
	nDependency : UINT;
	bAllSafe : BOOL;
	Snapshot : ST_ServiceExecutionSnapshot;
END_VAR
H_OnStopping := E_PackMLHookResult.Busy;
IF bFirstScan THEN M_ClearLifecycleRequests(); END_IF
IF NOT _OwnershipHeld THEN
	H_OnStopping := E_PackMLHookResult.Done;
	RETURN;
END_IF
bAllSafe := TRUE;
FOR nDependency := 1 TO _DependencyCount DO
	IF NOT M_GetDependencySnapshot(DependencyIndex := nDependency, Snapshot => Snapshot) THEN
		bAllSafe := FALSE;
		CONTINUE;
	END_IF
	CASE Snapshot.PackMLOut.eStateCurrent OF
		E_PackMLState.Idle, E_PackMLState.Stopped:
			;
		E_PackMLState.Aborted:
			M_AddError(MainErrorId := TO_UDINT(E_CompositeServiceErrorCode.ChildAbortedUnexpectedly),
				SourceErrorId := TO_UDINT(Snapshot.PackMLOut.eStateErrorID),
				Message := 'A Composite dependency aborted while stopping.');
			RequestCommand(eTargetCmd := E_PackMLCommand.Abort);
			RETURN;
	ELSE
		bAllSafe := FALSE;
		M_EnsureLifecycleCommand(DependencyIndex := nDependency, Command := E_PackMLCommand.Stop);
	END_CASE
END_FOR
IF bAllSafe THEN H_OnStopping := E_PackMLHookResult.Done; END_IF
END_METHOD

METHOD PROTECTED FINAL M_AddDependency : BOOL
VAR_INPUT
	ServiceId : UDINT;
END_VAR
M_AddDependency := FALSE;
IF NOT _DefinitionOpen THEN RETURN; END_IF
IF _DependencyCount >= Param_Config.MaxCompositeDependencies THEN
	_DependencyOverflow := TRUE;
	RETURN;
END_IF
_DependencyCount := _DependencyCount + 1;
_DependencyServiceIds[_DependencyCount] := ServiceId;
M_AddDependency := TRUE;
END_METHOD

METHOD PRIVATE M_ClearLifecycleRequests
MEMSET(ADR(_LifecycleCommandSubmitted), 0, SIZEOF(_LifecycleCommandSubmitted));
END_METHOD

METHOD PROTECTED FINAL M_CommandDependency : E_ServiceCallSubmitResult
VAR_INPUT
	ServiceId : UDINT;
	Command : E_PackMLCommand;
END_VAR
M_CommandDependency := _ServiceCaller.M_Command(ServiceId := ServiceId, Command := Command);
END_METHOD

METHOD PRIVATE M_EnsureLifecycleCommand
VAR_INPUT
	DependencyIndex : UINT;
	Command : E_PackMLCommand;
END_VAR
VAR
	SubmitResult : E_ServiceCallSubmitResult;
	CommandState : E_ServiceInternalCommandState;
END_VAR
IF (DependencyIndex = 0) OR (DependencyIndex > _DependencyCount) THEN RETURN; END_IF

// 對所有 Dependency Service 下統一命令
IF NOT _LifecycleCommandSubmitted[DependencyIndex] THEN
	SubmitResult := M_CommandDependency(ServiceId := _DependencyServiceIds[DependencyIndex], Command := Command);
	IF SubmitResult = E_ServiceCallSubmitResult.Queued THEN
		_LifecycleCommandSubmitted[DependencyIndex] := TRUE;
	ELSIF SubmitResult <> E_ServiceCallSubmitResult.Busy THEN
		_LifecycleCommandSubmitted[DependencyIndex] := TRUE;
		M_AddError(MainErrorId := TO_UDINT(E_CompositeServiceErrorCode.InternalCallSubmitFailed),
			SourceErrorId := TO_UDINT(SubmitResult), Message := 'A Composite cleanup command could not be queued.');
	END_IF
	RETURN;
END_IF

CommandState := M_GetDependencyCommandState(ServiceId := _DependencyServiceIds[DependencyIndex]);
IF CommandState = E_ServiceInternalCommandState.Rejected THEN
	M_AddError(MainErrorId := TO_UDINT(E_CompositeServiceErrorCode.InternalCommandRejected),
		SourceErrorId := TO_UDINT(Command), Message := 'A Composite cleanup command was rejected.');
END_IF
END_METHOD

METHOD PROTECTED FINAL M_FailSequence
VAR_INPUT
	ErrorCode : E_CompositeServiceErrorCode;
	FailedServiceId : UDINT;
	SourceErrorId : UDINT;
	Message : STRING;
END_VAR
VAR
	EffectiveErrorCode : E_CompositeServiceErrorCode;
	EffectiveSourceErrorId : UDINT;
END_VAR
_SequenceFailed := TRUE;
EffectiveErrorCode := ErrorCode;
EffectiveSourceErrorId := SourceErrorId;
IF EffectiveErrorCode = E_CompositeServiceErrorCode.None THEN
	EffectiveErrorCode := E_CompositeServiceErrorCode.SequenceFailed;
END_IF
IF EffectiveSourceErrorId = 0 THEN
	EffectiveSourceErrorId := FailedServiceId;
END_IF
M_AddError(MainErrorId := TO_UDINT(EffectiveErrorCode),
	SourceErrorId := EffectiveSourceErrorId, Message := Message);
END_METHOD

METHOD PROTECTED FINAL M_GetDependencyCommandState : E_ServiceInternalCommandState
VAR_INPUT
	ServiceId : UDINT;
END_VAR
M_GetDependencyCommandState := _ServiceCaller.M_GetCommandState(ServiceId := ServiceId);
END_METHOD

METHOD PROTECTED FINAL M_GetDependencyServiceSnapshot : BOOL
VAR_INPUT
	ServiceId : UDINT;
END_VAR
VAR_OUTPUT
	Snapshot : ST_ServiceExecutionSnapshot;
END_VAR
M_GetDependencyServiceSnapshot := _ServiceCaller.M_GetServiceSnapshot(
	ServiceId := ServiceId, Snapshot => Snapshot);
END_METHOD

METHOD PRIVATE M_GetDependencySnapshot : BOOL
VAR_INPUT
	DependencyIndex : UINT;
END_VAR
VAR_OUTPUT
	Snapshot : ST_ServiceExecutionSnapshot;
END_VAR
M_GetDependencySnapshot := FALSE;
MEMSET(ADR(Snapshot), 0, SIZEOF(Snapshot));
IF (DependencyIndex = 0) OR (DependencyIndex > _DependencyCount) THEN RETURN; END_IF
M_GetDependencySnapshot := M_GetDependencyServiceSnapshot(
	ServiceId := _DependencyServiceIds[DependencyIndex], Snapshot => Snapshot);
END_METHOD

METHOD PUBLIC FINAL M_RegisterDefinition : BOOL
VAR_INPUT
	CompositeServiceId : UDINT;
END_VAR
VAR_IN_OUT
	Coordinator : FB_ServiceCoordinator;
END_VAR
VAR
	nDependencyCount : UINT;
END_VAR
M_RegisterDefinition := FALSE;

IF _DefinitionAttempted THEN
	RETURN;
END_IF

_DefinitionAttempted := TRUE;

// Clear dependency services
MEMSET(ADR(_DependencyServiceIds), 0, SIZEOF(_DependencyServiceIds));
_DependencyCount := 0;
_DependencyOverflow := FALSE;

// Add dependency services
_DefinitionOpen := TRUE;
H_DeclareServices();
_DefinitionOpen := FALSE;

// Check the amount of dependency services
nDependencyCount := _DependencyCount;
IF _DependencyOverflow THEN
	nDependencyCount := Param_Config.MaxCompositeDependencies + 1;
END_IF

IF NOT Coordinator.M_RegisterCompositeDefinition(
	CompositeServiceId := CompositeServiceId,
	DependencyCount := nDependencyCount,
	DependencyIds := _DependencyServiceIds) THEN RETURN; END_IF

IF NOT _ServiceCaller.M_Configure(
	CallerServiceId := CompositeServiceId,
	Coordinator := Coordinator) THEN RETURN; END_IF

_Coordinator REF= Coordinator;
_Configured := TRUE;
M_RegisterDefinition := TRUE;
END_METHOD

METHOD PROTECTED FINAL M_StartDependency : E_ServiceCallSubmitResult
VAR_INPUT
	ServiceId : UDINT;
	Parameters : ANY;
END_VAR
M_StartDependency := _ServiceCaller.M_Start(ServiceId := ServiceId, Parameters := Parameters);
END_METHOD

METHOD PROTECTED FINAL M_UpdateCompositeService
M_UpdateService(CompletionBehavior := E_ServiceCompletionBehavior.NaturalCompletion);
END_METHOD

END_FUNCTION_BLOCK

// ---- POUs/20_Service/FB_ServiceBase.TcPOU
{attribute 'reflection'}
FUNCTION_BLOCK FB_ServiceBase EXTENDS FB_PackMLModeSet
VAR_INPUT
	Ctrl : REFERENCE TO ST_ServiceCtrl;
	Context : REFERENCE TO ST_ServiceContext;
	
	// The Module assigns a unique ID to this Service instance.
	ServiceId : T_ResourceOwnerId;
END_VAR

VAR_OUTPUT
	Status : ST_ServiceStatus;
END_VAR

VAR
	_CmdRequestOneShot : R_TRIG;
	_LastObservedPackMLState : E_PackMLState := E_PackMLState.Undefined;
	_ActiveExecuteSubStateRecord : UINT;
	
	{attribute 'instance-path'}
    {attribute 'noinit'}
	_Path : STRING;
END_VAR

METHOD PROTECTED H_GetExecuteSubState : UDINT
H_GetExecuteSubState := 0;
END_METHOD

METHOD PROTECTED H_GetExecuteSubStateName : STRING(80)
H_GetExecuteSubStateName := '';
END_METHOD

METHOD PROTECTED FINAL M_AddError : BOOL
VAR_INPUT
	MainErrorId : UDINT;
	SourceErrorId : UDINT;
	Message : STRING;
END_VAR

VAR
	nIndex : UINT;
	nFirstEmpty : UINT;
END_VAR
M_AddError := FALSE;
nFirstEmpty := 0;

FOR nIndex := 1 TO Param_Config.MaxServiceError DO
	IF Status.ErrorList[nIndex].MainErrorId = 0 THEN
		IF nFirstEmpty = 0 THEN
			nFirstEmpty := nIndex;
			EXIT;
		END_IF

	ELSIF Status.ErrorList[nIndex].MainErrorId = MainErrorId THEN
		// The same error event is already recorded for this task cycle.
		RETURN;
	END_IF
END_FOR

// Preserve the first ten errors; reject new errors when the list is full.
IF nFirstEmpty = 0 THEN
	RETURN;
END_IF

Status.ErrorList[nFirstEmpty].ModuleId := Context.ModuleId;
Status.ErrorList[nFirstEmpty].ServiceId := ServiceId;
Status.ErrorList[nFirstEmpty].MainErrorId := MainErrorId;
Status.ErrorList[nFirstEmpty].SourceErrorId := SourceErrorId;
Status.ErrorList[nFirstEmpty].Message := Message;
Status.ErrorList[nFirstEmpty].Path := _Path;
Status.ErrorList[nFirstEmpty].Severity := E_Severity.Alarm;
Status.ErrorList[nFirstEmpty].DateTime := Context.UtcDateTime;
Status.ErrorList[nFirstEmpty].Active := TRUE;
Status.ErrorList[nFirstEmpty].Acknowledged := FALSE;
Status.ErrorList[nFirstEmpty].OccurrenceCount := 1;
M_AddError := TRUE;
END_METHOD

METHOD PROTECTED FINAL M_ClearAllData
MEMSET(ADR(Status.Data), 0, SIZEOF(Status.Data));
END_METHOD

METHOD PROTECTED FINAL M_ClearAllError : BOOL
VAR_INPUT
END_VAR
MEMSET(ADR(Status.ErrorList), 0, SIZEOF(Status.ErrorList));
M_ClearAllError := TRUE;
END_METHOD

METHOD PROTECTED FINAL M_ClearData : BOOL
VAR_INPUT
	DataId : UDINT;
END_VAR
VAR
	nIndex : UINT;
END_VAR
M_ClearData := FALSE;
IF DataId = 0 THEN
	RETURN;
END_IF

FOR nIndex := 1 TO Param_Config.MaxServiceData DO
	IF Status.Data.DataList[nIndex].Id = DataId THEN
		MEMSET(ADR(Status.Data.DataList[nIndex]), 0, SIZEOF(Status.Data.DataList[nIndex]));
		IF Status.Data.Count > 0 THEN
			Status.Data.Count := Status.Data.Count - 1;
		END_IF
		Status.Data.Overflow := FALSE;
		M_ClearData := TRUE;
		RETURN;
	END_IF
END_FOR
END_METHOD

METHOD PRIVATE M_ClearExecuteSubStateStatus
MEMSET(ADR(Status.ExecuteSubState), 0, SIZEOF(Status.ExecuteSubState));
_ActiveExecuteSubStateRecord := 0;
END_METHOD

METHOD PRIVATE M_CloseExecuteSubStateRecord
IF (_ActiveExecuteSubStateRecord > 0)
	AND (_ActiveExecuteSubStateRecord <= Status.ExecuteSubState.RecordCount) THEN
	Status.ExecuteSubState.Records[_ActiveExecuteSubStateRecord].EndTimestamp := Context.UtcDateTime;
END_IF
_ActiveExecuteSubStateRecord := 0;
END_METHOD

METHOD PROTECTED FINAL M_UpdateData : BOOL
VAR_INPUT
	DataId : UDINT;
	Name : STRING(30);
	DataType : E_DescriptorType;
	Unit : STRING(10);
	Value : STRING(80);
END_VAR
VAR
	nIndex : UINT;
	nTargetIndex : UINT;
	nFirstEmpty : UINT;
END_VAR
M_UpdateData := FALSE;
IF DataId = 0 THEN
	RETURN;
END_IF

nTargetIndex := 0;
nFirstEmpty := 0;
FOR nIndex := 1 TO Param_Config.MaxServiceData DO
	IF Status.Data.DataList[nIndex].Id = DataId THEN
		nTargetIndex := nIndex;
		EXIT;
	ELSIF (Status.Data.DataList[nIndex].Id = 0) AND (nFirstEmpty = 0) THEN
		nFirstEmpty := nIndex;
	END_IF
END_FOR

IF nTargetIndex = 0 THEN
	IF nFirstEmpty = 0 THEN
		Status.Data.Overflow := TRUE;
		RETURN;
	END_IF
	nTargetIndex := nFirstEmpty;
	Status.Data.Count := Status.Data.Count + 1;
END_IF

Status.Data.DataList[nTargetIndex].Id := DataId;
Status.Data.DataList[nTargetIndex].Name := Name;
Status.Data.DataList[nTargetIndex].DataType := DataType;
Status.Data.DataList[nTargetIndex].Unit := Unit;
Status.Data.DataList[nTargetIndex].Value := Value;
M_UpdateData := TRUE;
END_METHOD

METHOD PRIVATE M_UpdateExecuteSubStateStatus
VAR_INPUT
	ExecuteActionEvaluated : BOOL;
END_VAR
VAR
	NewState : UDINT;
	NewRecordIndex : UINT;
END_VAR
IF PackMLOut.eStateCurrent <> E_PackMLState.Execute THEN
	M_CloseExecuteSubStateRecord();
	Status.ExecuteSubState.CurrentStep := 0;
	RETURN;
END_IF

// Entering Execute does not run H_OnExecute until the following Service scan.
// Do not sample a substate until an Execute action has actually been evaluated.
IF NOT ExecuteActionEvaluated THEN
	M_CloseExecuteSubStateRecord();
	Status.ExecuteSubState.CurrentStep := 0;
	RETURN;
END_IF

NewState := H_GetExecuteSubState();
IF NewState = Status.ExecuteSubState.CurrentStep THEN
	RETURN;
END_IF

M_CloseExecuteSubStateRecord();
Status.ExecuteSubState.CurrentStep := NewState;

// State zero means that the Service currently exposes no Execute substate.
IF NewState = 0 THEN
	RETURN;
END_IF

// Preserve the first records. CurrentState continues to update after overflow.
IF Status.ExecuteSubState.RecordCount >= Param_Config.MaxExecuteSubStateRecords THEN
	Status.ExecuteSubState.Overflow := TRUE;
	RETURN;
END_IF

NewRecordIndex := Status.ExecuteSubState.RecordCount + 1;
Status.ExecuteSubState.RecordCount := NewRecordIndex;
Status.ExecuteSubState.Records[NewRecordIndex].Step := NewState;
Status.ExecuteSubState.Records[NewRecordIndex].Name := H_GetExecuteSubStateName();
Status.ExecuteSubState.Records[NewRecordIndex].StartTimestamp := Context.UtcDateTime;
Status.ExecuteSubState.Records[NewRecordIndex].EndTimestamp := '';
_ActiveExecuteSubStateRecord := NewRecordIndex;
END_METHOD

METHOD PROTECTED FINAL M_UpdateService
VAR_INPUT
	CompletionBehavior : E_ServiceCompletionBehavior;
END_VAR
VAR
	bEnteredStarting : BOOL;
	PreviousPackMLState : E_PackMLState;
END_VAR
PreviousPackMLState := PackMLOut.eStateCurrent;
PackMLIn := Ctrl.PackMLIn;
SUPER^();

_CmdRequestOneShot(CLK:= PackMLIn.bCommandChangeRequest, Q=> );

// Starting may complete and enter Execute in the same scan. In that case,
// eStatePrevious still exposes the transient Starting state.
bEnteredStarting :=
	// Starting 執行超過1個 scan
	((PackMLOut.eStateCurrent = E_PackMLState.Starting)
		AND (_LastObservedPackMLState <> E_PackMLState.Starting))

	// Starting 在同一scan 就結束，即 _LastObservedPackMLState = Idle & PackMLOut.eStateCurrent = Execute
	OR ((PackMLOut.eStateCurrent = E_PackMLState.Execute)
		AND (PackMLOut.eStatePrevious = E_PackMLState.Starting)
		AND (_LastObservedPackMLState <> E_PackMLState.Starting)
		AND (_LastObservedPackMLState <> E_PackMLState.Execute));

IF bEnteredStarting THEN
	M_ClearExecuteSubStateStatus();
END_IF

// Update status.
Status.PackMLOut := PackMLOut;
M_UpdateExecuteSubStateStatus(
	ExecuteActionEvaluated := PreviousPackMLState = E_PackMLState.Execute);
Status.CompletionBehavior := CompletionBehavior;
Status.ServiceId := ServiceId;
IF _CmdRequestOneShot.Q THEN // Acknowledge to upper controller that command received
	Status.ResponseId := Ctrl.RequestId;
END_IF

_LastObservedPackMLState := PackMLOut.eStateCurrent;
END_METHOD

END_FUNCTION_BLOCK

// ---- POUs/30_PackML_Base/FB_PackMLModeSet.TcPOU
FUNCTION_BLOCK FB_PackMLModeSet EXTENDS FB_PackMLBase
VAR_INPUT
END_VAR
VAR_OUTPUT
END_VAR
VAR
END_VAR

SUPER^();

METHOD PROTECTED FINAL H_IsCommandAllowedByMode : BOOL
VAR_INPUT
	eRequestedCommand	: E_PackMLCommand;
	eActiveMode	: T_PackMLMode;
END_VAR
CASE eActiveMode OF
	E_PackMLMode.Manual:
		// Supported commands in manual mode
		CASE eRequestedCommand OF
			E_PackMLCommand.Reset,
			E_PackMLCommand.Start,
			E_PackMLCommand.Stop,
			E_PackMLCommand.Abort,
			E_PackMLCommand.Clear:
				H_IsCommandAllowedByMode := TRUE;
			ELSE
				H_IsCommandAllowedByMode := FALSE;
		END_CASE
	
	E_PackMLMode.Production,
	E_PackMLMode.Unknown:
		// Support all commands in production mode
		H_IsCommandAllowedByMode := TRUE;
END_CASE
END_METHOD

METHOD PROTECTED FINAL H_IsModeSupported : BOOL
VAR_INPUT
	eRequestedMode	: T_PackMLMode;
END_VAR
CASE eRequestedMode OF
	E_PackMLMode.Manual,
	E_PackMLMode.Production:
		H_IsModeSupported := TRUE;

	ELSE
		H_IsModeSupported := FALSE;
END_CASE
END_METHOD

METHOD PROTECTED FINAL H_IsStateSupportedByMode : BOOL
VAR_INPUT
	eRequestedMode	: T_PackMLMode;
	eCurrentState	: E_PackMLState;
END_VAR
CASE eRequestedMode OF
	
	E_PackMLMode.Manual:
		// Support states in manual mode
		CASE eCurrentState OF
			E_PackMLState.Idle,
			E_PackMLState.Starting,
			E_PackMLState.Execute,
			E_PackMLState.Aborting,
			E_PackMLState.Aborted,
			E_PackMLState.Clearing,
			E_PackMLState.Stopped,
			E_PackMLState.Resetting:
			H_IsStateSupportedByMode := TRUE;
			
			ELSE
				H_IsStateSupportedByMode := FALSE;
		END_CASE
		
	
	E_PackMLMode.Production,
	E_PackMLMode.Unknown:
		// Support all state in production mode
		H_IsStateSupportedByMode := TRUE;
END_CASE
END_METHOD

END_FUNCTION_BLOCK

// ---- POUs/20_Service/Material Service/FB_SetMaterialService.TcPOU
FUNCTION_BLOCK FB_SetMaterialService EXTENDS FB_ServiceBase
VAR_INPUT
	Param : ST_MaterialParam;
END_VAR

VAR_IN_OUT
	WaferStatusList : ARRAY[*] OF ST_WaferStatus; 
END_VAR

VAR
	_ActiveParam : ST_MaterialParam;
	_TargetIndex : DINT;
END_VAR

M_UpdateService(CompletionBehavior := E_ServiceCompletionBehavior.NaturalCompletion);

METHOD PROTECTED H_OnExecute : E_PackMLHookResult
VAR_INPUT
	bFirstScan	: BOOL;
END_VAR

VAR
	nIndex : DINT;
END_VAR
H_OnExecute := E_PackMLHookResult.Busy;

CASE _ActiveParam.CmdType OF
	E_SetMaterialCmdType.Modify:
		WaferStatusList[_TargetIndex].MaterialContext.Id := _ActiveParam.MaterialId;
		WaferStatusList[_TargetIndex].MaterialContext.OperationState := _ActiveParam.MaterialOperateState;

	E_SetMaterialCmdType.Clear:
		MEMSET(
			ADR(WaferStatusList[_TargetIndex].MaterialContext),
			0,
			SIZEOF(WaferStatusList[_TargetIndex].MaterialContext));

	E_SetMaterialCmdType.ClearAll:
		FOR nIndex := LOWER_BOUND(WaferStatusList, 1)
			TO UPPER_BOUND(WaferStatusList, 1) DO
			MEMSET(
				ADR(WaferStatusList[nIndex].MaterialContext),
				0,
				SIZEOF(WaferStatusList[nIndex].MaterialContext));
		END_FOR

	ELSE
		// Starting validates and snapshots the command. This is a defensive guard.
		M_AddError(
			MainErrorId := TO_UDINT(E_FrameworkServiceErrorCode.SetMaterial_InvalidCmd),
			SourceErrorId := 0,
			Message := 'The snapshotted material command is invalid.');
		RequestCommand(E_PackMLCommand.Stop);
		RETURN;
END_CASE

H_OnExecute := E_PackMLHookResult.Done;
END_METHOD

METHOD PROTECTED H_OnStarting : E_PackMLHookResult
VAR_INPUT
	bFirstScan	: BOOL;
END_VAR

VAR
	nIndex : DINT;
	nTargetMatchCount : UINT;
END_VAR
H_OnStarting := E_PackMLHookResult.Busy;

IF bFirstScan THEN
	// Execute must use the same values that were validated during Starting.
	_ActiveParam := Param;
	_TargetIndex := 0;
END_IF

CASE _ActiveParam.CmdType OF
	E_SetMaterialCmdType.Modify,
	E_SetMaterialCmdType.Clear:
		IF _ActiveParam.TargetEndpointId = 0 THEN
			M_AddError(
				MainErrorId := TO_UDINT(E_FrameworkServiceErrorCode.SetMaterial_TaEpIdRequired),
				SourceErrorId := 0,
				Message := 'TargetEndpointId must be non-zero for Modify or Clear.');
			RequestCommand(E_PackMLCommand.Stop);
			RETURN;
		END_IF

		nTargetMatchCount := 0;
		FOR nIndex := LOWER_BOUND(WaferStatusList, 1)
			TO UPPER_BOUND(WaferStatusList, 1) DO
			IF WaferStatusList[nIndex].EndpointId = _ActiveParam.TargetEndpointId THEN
				nTargetMatchCount := nTargetMatchCount + 1;
				_TargetIndex := nIndex;
			END_IF
		END_FOR

		IF nTargetMatchCount = 0 THEN
			M_AddError(
				MainErrorId := TO_UDINT(E_FrameworkServiceErrorCode.SetMaterial_TaEpNotFound),
				SourceErrorId := 0,
				Message := 'TargetEndpointId was not found in WaferStatusList.');
			RequestCommand(E_PackMLCommand.Stop);
			RETURN;
		END_IF

		IF nTargetMatchCount > 1 THEN
			M_AddError(
				MainErrorId := TO_UDINT(E_FrameworkServiceErrorCode.SetMaterial_DuplicateTaEpId),
				SourceErrorId := 0,
				Message := 'TargetEndpointId is duplicated in WaferStatusList.');
			RequestCommand(E_PackMLCommand.Stop);
			RETURN;
		END_IF

	E_SetMaterialCmdType.ClearAll:
		// ClearAll intentionally ignores TargetEndpointId and MaterialContext.
		_TargetIndex := 0;

	ELSE
		M_AddError(
			MainErrorId := TO_UDINT(E_FrameworkServiceErrorCode.SetMaterial_InvalidCmd),
			SourceErrorId := 0,
			Message := 'CmdType is not a supported material command.');
		RequestCommand(E_PackMLCommand.Stop);
		RETURN;
END_CASE

H_OnStarting := E_PackMLHookResult.Done;
END_METHOD

END_FUNCTION_BLOCK

// ---- POUs/FB_UtcClock.TcPOU
FUNCTION_BLOCK FB_UtcClock
VAR_OUTPUT
	UtcDateTime : STRING(20);
END_VAR

VAR
	_UtcFileTime : T_FILETIME64;
	_UtcSystemTime : TIMESTRUCT;
	_FormattedDateTime : STRING(24);
END_VAR

_UtcFileTime := F_GetSystemTime();
_UtcSystemTime := FILETIME64_TO_SYSTEMTIME(_UtcFileTime);
_FormattedDateTime := SYSTEMTIME_TO_STRING(_UtcSystemTime);

// SYSTEMTIME_TO_STRING returns YYYY-MM-DD-hh:mm:ss.xxx.
// Publish a compact, fixed-width UTC timestamp: YYYYMMDDHHMMSSUUU.
UtcDateTime := CONCAT(LEFT(_FormattedDateTime, 4), MID(_FormattedDateTime, 2, 6));
UtcDateTime := CONCAT(UtcDateTime, MID(_FormattedDateTime, 2, 9));
UtcDateTime := CONCAT(UtcDateTime, MID(_FormattedDateTime, 2, 12));
UtcDateTime := CONCAT(UtcDateTime, MID(_FormattedDateTime, 2, 15));
UtcDateTime := CONCAT(UtcDateTime, MID(_FormattedDateTime, 2, 18));
UtcDateTime := CONCAT(UtcDateTime, MID(_FormattedDateTime, 3, 21));

END_FUNCTION_BLOCK
